// Data types/Touch Probe/E_SignalSource
TYPE E_SignalSource :
 (
	SignalSource_Default,			(* predefined or externally configured *)
	SignalSource_Input1,			(* not selectable in most cases! - digital drive input 1 - from TC 2.11 NC driver 2014 and not TOUCHPROBEMODE_SINGLE_COMPATIBILITYMODE *)
	SignalSource_Input2,			(* not selectable in most cases! - digital drive input 2 - from TC 2.11 NC driver 2014 and not TOUCHPROBEMODE_SINGLE_COMPATIBILITYMODE *)
	SignalSource_Input3,			(* not selectable in most cases! - digital drive input 3 - from TC 2.11 NC driver 2014 and not TOUCHPROBEMODE_SINGLE_COMPATIBILITYMODE *)
	SignalSource_Input4,			(* not selectable in most cases! - digital drive input 4 - from TC 2.11 NC driver 2014 and not TOUCHPROBEMODE_SINGLE_COMPATIBILITYMODE *)
	SignalSource_ZeroPulse := 128,	(* encoder zero pulse. Availability depending on hardware - from TC 2.11 NC driver 2014 and not TOUCHPROBEMODE_SINGLE_COMPATIBILITYMODE *)
	SignalSource_DriveDefined		(* defined by drive parameters - e. g. CAN object 0x60D0 - from TC 2.11 NC driver 2014 and not TOUCHPROBEMODE_SINGLE_COMPATIBILITYMODE *)
 ) UINT;
END_TYPE

// Data types/Touch Probe/E_TouchProbe
(* MC_TouchProbe probes *)
TYPE E_TouchProbe :
 (
	TouchProbe1 := 1,	(* first hardware probe unit with AX2000, SERCOS, KL5xxx and others *)
	TouchProbe2,		(* 2nd probe unit - available from MC_TouchProbe V2 *)
	TouchProbe3,		(* 3rd probe unit - available from MC_TouchProbe V2 *)
	TouchProbe4,		(* 4th probe unit - available from MC_TouchProbe V2 *)
	PlcEvent := 10		(* simple PLC signal TRUE/FALSE *)
 ) UINT;
END_TYPE

// Data types/Touch Probe/E_TouchProbeMode
TYPE E_TouchProbeMode :
 (
	TOUCHPROBEMODE_SINGLE_COMPATIBILITYMODE, (* for TC 2.10 and 2.11 till NC driver 2013 / legacy interface*)
	TOUCHPROBEMODE_SINGLE,			(* multi probe interface - from 2.11 NC driver 2014 / new interface *)
	TOUCHPROBEMODE_CONTINOUS		(* multi probe interface - from 2.11 NC driver 2014 / new interface *)
 ) UINT;
END_TYPE

// Data types/Touch Probe/MC_TouchProbeRecordedData
TYPE MC_TouchProbeRecordedData :
STRUCT
	Counter : LREAL;
	RecordedPosition : LREAL;
	AbsolutePosition	: LREAL;
	ModuloPosition 	: LREAL;
END_STRUCT
END_TYPE

// Data types/Touch Probe/TRIGGER_REF
TYPE TRIGGER_REF :
STRUCT
	EncoderID  		: UDINT;				(* 1..255 *)
	TouchProbe 		: E_TouchProbe;		(* probe unit definition *)
	SignalSource	: E_SignalSource;		(* optional physical signal source used by the probe unit - from TC 2.11 NC driver 2014 with MC_TouchProbe_V2 / no effect for old implementation or TOUCHPROBEMODE_SINGLE_COMPATIBILITYMODE *)
	Edge 			: E_SignalEdge;		(* rising or falling signal edge *)
	(* Mode=TOUCHPROBEMODE_SINGLE as default - changed from TC3 - 2013-04-09 KSt *)
	Mode			: E_TouchProbeMode := TOUCHPROBEMODE_SINGLE; 	(* single shot or continuous monitoring - available from TwinCAT 2.11 NC driver 2014 with MC_TouchProbe_V2 *)
	PlcEvent 		: BOOL;				(* PLC trigger signal input when TouchProbe (probe unit) is set to 'PlcEvent' *)
	ModuloPositions : BOOL;			(* interpretation of FirstPosition, LastPosition and RecordedPosition as modulo positions when TRUE *)
{attribute 'conditionalshow'}
	ProbeState 		: _E_TouchProbeState;	(* internal state of the touch probe sequence *)
END_STRUCT
END_TYPE

// POUs/[Internal]/Objects/_FBAXIS_REF
{attribute 'conditionalshow'}
TYPE _FBAXIS_REF : AXIS_REF;
END_TYPE

// Global Variables/Global_Variables
VAR_GLOBAL
	TcMcGlobal : _TCMCGLOBAL;
END_VAR
VAR_GLOBAL CONSTANT
	DEFAULT_HOME_POSITION 	:	LREAL 	:= 1.0E307;
	DEFAULT_BACKLASHVALUE 	: 	LREAL 	:= 1.0E307;
END_VAR

// Version/Global_Version
{attribute 'TcGenerated'}
{attribute 'no-analysis'}
{attribute 'linkalways'}
// This function has been automatically generated from the project information.
VAR_GLOBAL CONSTANT
	{attribute 'const_non_replaced'}
	stLibVersion_Tc2_MC2 : ST_LibVersion := (iMajor := 3, iMinor := 3, iBuild := 54, iRevision := 0, nFlags := 1, sVersion := '3.3.54.0');
END_VAR

// Data types/Axis Reference/AXIS_REF
(*
	AXIS_REF data structure

	The FBAXIS_REF is actually not a function block but a data structure
	It includes the axis I/O variables as well as additional information.
	The reason for not using a STRUCT is that structures cannot hold
	located I/O variables.
	The user is supposed to use the AXIS_REF data type which internally
	redirects the type to this function block definition (alias).
*)
{attribute 'conditionalshow_all_locals'}
FUNCTION_BLOCK AXIS_REF
VAR_INPUT
	PlcToNc   AT %Q* : PLCTONC_AXIS_REF;
END_VAR
VAR_OUTPUT
	NcToPlc   AT %I* : NCTOPLC_AXIS_REF;
	ADS              : ST_AdsAddress;
	Status           : ST_AxisStatus;
END_VAR
VAR_INPUT
	DriveAddress		: ST_DriveAddress;
END_VAR
VAR
	_internal : _InternalAxisRefData;
	Storage				:	ARRAY [0..127] OF DWORD;	(* universal storage for internal use *)
END_VAR


ReadStatus();

ACTION ReadStatus:
(* NC cycle counter will be incremented after NC task updated the NcToPlc data structure *)
_internal.NcCycleCounter_AtReadStatusCall := SHR(NcToPlc.OpModeDWord, 24);

(* avoid multiple updates during one cycle which would cause additional CPU load *)
IF _internal.NcCycleCounter_AtReadStatusCall <> Status.NcCycleCounter OR _internal.NcCycleCounter_AtReadStatusCall=0 THEN

	(* new cycle - call status function *)
	_internal.LastTaskIndex_AtReadStatusCall := Status.UpdateTaskIndex;

	(* update the axis status
		ForceTaskIndexUpdate makes sure that the index of the current  task will be updated. 
		ForceTaskIndexUpdate=false saves time because a system call to gettaskindex will be avoided.
	*)
	Status := _F_ReadStatus( ForceTaskIndexUpdate:=_internal.CounterSameTaskIndex_AtReadStatusCall<100, NcToPlc := NcToPlc, PlcToNc := PlcToNc, LastStatus:=Status );

	DriveAddress.TcAxisObjectId := _F_GetTcAxisObjectId(AxisId := NcToPlc.AxisId);
	
	(* count number of cycles with the same task index *)
	IF _internal.LastTaskIndex_AtReadStatusCall=Status.UpdateTaskIndex THEN
		IF _internal.CounterSameTaskIndex_AtReadStatusCall<100 THEN
			(* increment counter as long as the update task index does not change - max value is 100 *)
			_internal.CounterSameTaskIndex_AtReadStatusCall := _internal.CounterSameTaskIndex_AtReadStatusCall + 1;
		END_IF
	ELSE
		(* reset counter since update task index has changed - this is not supposed to happen but a user might call ReadStatus in several tasks *)
		_internal.CounterSameTaskIndex_AtReadStatusCall:= 0;
	END_IF
END_IF
END_ACTION

END_FUNCTION_BLOCK

// POUs/[Internal]/_F_ReadStatus
{attribute 'conditionalshow'}
FUNCTION _F_ReadStatus : ST_AxisStatus
VAR_INPUT
	ForceTaskIndexUpdate : BOOL; (* force update of the taskindex with GETCURTASKINDEX - otherwise update only once - 20100416 KSt *)
END_VAR
VAR_IN_OUT
	NcToPlc : NCTOPLC_AXIS_REF;
	PlcToNc : PLCTONC_AXIS_REF;
	LastStatus : ST_AxisStatus;
END_VAR
VAR
	GetTaskIndex : GETCURTASKINDEX;
END_VAR

 (* MOTION CONTROL STATEMACHINE STATES *)
(* no need to initialize since function result is already intialized - 20100416 KSt *)
(*
_F_ReadStatus.ErrorStop			:= FALSE;
_F_ReadStatus.Disabled 			:= FALSE;
_F_ReadStatus.Stopping			:= FALSE;
_F_ReadStatus.StandStill			:= FALSE;
_F_ReadStatus.DiscreteMotion		:= FALSE;
_F_ReadStatus.ContinuousMotion	:= FALSE;
_F_ReadStatus.SynchronizedMotion	:= FALSE;
_F_ReadStatus.Homing			:= FALSE;
*)

_F_ReadStatus.MotionState := _F_AxisState(NcToPlc, PlcToNc);
CASE _F_ReadStatus.MotionState OF
	MC_AXISSTATE_DISABLED :
		_F_ReadStatus.Disabled := TRUE;
	MC_AXISSTATE_STANDSTILL :
		_F_ReadStatus.StandStill := TRUE;
	MC_AXISSTATE_ERRORSTOP :
		_F_ReadStatus.ErrorStop := TRUE;
	MC_AXISSTATE_STOPPING :
		_F_ReadStatus.Stopping := TRUE;
	MC_AXISSTATE_HOMING :
		_F_ReadStatus.Homing	:= TRUE;
	MC_AXISSTATE_DISCRETEMOTION :
		_F_ReadStatus.DiscreteMotion := TRUE;
	MC_AXISSTATE_CONTINOUSMOTION :
		_F_ReadStatus.ContinuousMotion := TRUE;
	MC_AXISSTATE_SYNCHRONIZEDMOTION :
		_F_ReadStatus.SynchronizedMotion := TRUE;
END_CASE

(* NcToPlc.StateDWord *)
_F_ReadStatus.Operational				:= NcToPlc.StateDWord.0;
_F_ReadStatus.Homed				:= NcToPlc.StateDWord.1;		(* homed *)
_F_ReadStatus.NotMoving				:= NcToPlc.StateDWord.2;
_F_ReadStatus.InPositionArea			:= NcToPlc.StateDWord.3;
_F_ReadStatus.inTargetPosition 		:= NcToPlc.StateDWord.4;
_F_ReadStatus.ProtectedMode				:= NcToPlc.StateDWord.5;
_F_ReadStatus.ErrorPropagationDelayed	:= NcToPlc.StateDWord.6;
_F_ReadStatus.HasBeenStopped		:= NcToPlc.StateDWord.7;
_F_ReadStatus.HasJob				:= NcToPlc.StateDWord.8;
_F_ReadStatus.Moving				:= NcToPlc.StateDWord.9 OR NcToPlc.StateDWord.10;
_F_ReadStatus.PositiveDirection		:= NcToPlc.StateDWord.9;
_F_ReadStatus.NegativeDirection 		:= NcToPlc.StateDWord.10;
_F_ReadStatus.HomingBusy			:= NcToPlc.StateDWord.11; 	(* homing *)
_F_ReadStatus.ConstantVelocity 		:= NcToPlc.StateDWord.12;
_F_ReadStatus.Compensating			:= NcToPlc.StateDWord.13;	(* superposition active *)
_F_ReadStatus.ExtSetPointGenEnabled 	:= NcToPlc.StateDWord.14;
_F_ReadStatus.PhasingActive 	:= NcToPlc.StateDWord.15;
_F_ReadStatus.ExternalLatchValid		:= NcToPlc.StateDWord.16;
_F_ReadStatus.NewTargetPosition		:= NcToPlc.StateDWord.17;
_F_ReadStatus.DriveLimitActive 	:= NcToPlc.StateDWord.18; (* 201801213 Fap *)
(*_F_ReadStatus.MovingEndless 		:= NcToPlc.StateDWord.19;	see continuous motion *)
_F_ReadStatus.ControlLoopClosed 		:= NcToPlc.StateDWord.20;
_F_ReadStatus.CamTableQueued 		:= NcToPlc.StateDWord.21;
_F_ReadStatus.CamDataQueued		:= NcToPlc.StateDWord.22;
_F_ReadStatus.CamScalingPending 		:= NcToPlc.StateDWord.23;
_F_ReadStatus.CmdBuffered	 		:= NcToPlc.StateDWord.24;
_F_ReadStatus.PTPmode	 			:= NcToPlc.StateDWord.25;
_F_ReadStatus.SoftLimitMinExceeded	:= NcToPlc.StateDWord.26;
_F_ReadStatus.SoftLimitMaxExceeded	:= NcToPlc.StateDWord.27;
_F_ReadStatus.DriveDeviceError	 	:= NcToPlc.StateDWord.28;
_F_ReadStatus.MotionCommandsLocked	:= NcToPlc.StateDWord.29;
_F_ReadStatus.IoDataInvalid			:= NcToPlc.StateDWord.30;
_F_ReadStatus.Error 					:= NcToPlc.StateDWord.31;

(* NcToPlc.nCoupleState *)
_F_ReadStatus.Coupled		:= NcToPlc.CoupleState > 1;

(* additional status data structue *)
_F_ReadStatus.ErrorID			:= NcToPlc.ErrorCode;
_F_ReadStatus.Accelerating 	:= NcToPlc.AxisState = INT_TO_DWORD(TCNC_PHASE_ACCPOS);
_F_ReadStatus.Decelerating 	:= NcToPlc.AxisState = INT_TO_DWORD(TCNC_PHASE_ACCNEG);

(* axis operation modes *)
_F_ReadStatus.OpMode.PositionAreaMonitoring	:= NcToPlc.OpModeDWord.0;
_F_ReadStatus.OpMode.TargetPositionMonitoring	:= NcToPlc.OpModeDWord.1;
_F_ReadStatus.OpMode.LoopMode				:= NcToPlc.OpModeDWord.2;
_F_ReadStatus.OpMode.MotionMonitoring		:= NcToPlc.OpModeDWord.3;
_F_ReadStatus.OpMode.PEHTimeMonitoring		:= NcToPlc.OpModeDWord.4;
_F_ReadStatus.OpMode.BacklashCompensation	:= NcToPlc.OpModeDWord.5;
_F_ReadStatus.OpMode.DelayedErrorReaction	:= NcToPlc.OpModeDWord.6;	(* 2008-02-20 KSt *)
_F_ReadStatus.OpMode.Modulo				:= NcToPlc.OpModeDWord.7;
_F_ReadStatus.OpMode.SimulationAxis			:= NcToPlc.OpModeDWord.8;	(* 2011-05-31 KSt *)
_F_ReadStatus.OpMode.StopMonitoring			:= NcToPlc.OpModeDWord.12;	(* 2011-12-09 KSt *)
_F_ReadStatus.OpMode.PositionLagMonitoring	:= NcToPlc.OpModeDWord.16;
_F_ReadStatus.OpMode.VelocityLagMonitoring	:= NcToPlc.OpModeDWord.17;
_F_ReadStatus.OpMode.SoftLimitMinMonitoring	:= NcToPlc.OpModeDWord.18;
_F_ReadStatus.OpMode.SoftLimitMaxMonitoring	:= NcToPlc.OpModeDWord.19;
_F_ReadStatus.OpMode.PositionCorrection		:= NcToPlc.OpModeDWord.20;
_F_ReadStatus.OpMode.AllowSlaveCommands	:= NcToPlc.OpModeDWord.21;	(* 2009-02-20 KSt *)
_F_ReadStatus.OpMode.AllowExtSetAxisCommands := NcToPlc.OpModeDWord.22;(* 2011-10-13 KSt *)
(* additional status bits in operation mode dword *)
_F_ReadStatus.NcApplicationRequest			:= NcToPlc.OpModeDWord.23;	(* 2010-04-06 KSt *)

(* NC cycle counter will be incremented after NC task updated the NcToPlc data structure *)
_F_ReadStatus.NcCycleCounter := SHR(NcToPlc.OpModeDWord, 24);

IF 	LastStatus.UpdateTaskIndex=0 OR ForceTaskIndexUpdate THEN
	GetTaskIndex(); (* function call causes high CPU load - supposed to be avoided - 20100416 KSt *)
	_F_ReadStatus.UpdateTaskIndex := GetTaskIndex.index;
	_F_ReadStatus.CycleCounter := TwinCAT_SystemInfoVarList._TaskInfo[_F_ReadStatus.UpdateTaskIndex].cycleCount;
	(*_F_ReadStatus.UpdateCycleTime := TwinCAT_SystemInfoVarList._TaskInfo[_F_ReadStatus.UpdateTaskIndex].cycleTime / LREAL#1.0E6;*)	(* Correction 2009-11-26 KSt *)
	_F_ReadStatus.UpdateCycleTime := TwinCAT_SystemInfoVarList._TaskInfo[_F_ReadStatus.UpdateTaskIndex].cycleTime / LREAL#1.0E7;	(* Correction 2014-05-20 KSt *)
ELSE
	_F_ReadStatus.UpdateTaskIndex := LastStatus.UpdateTaskIndex;
	_F_ReadStatus.CycleCounter := TwinCAT_SystemInfoVarList._TaskInfo[LastStatus.UpdateTaskIndex].cycleCount;
	(*_F_ReadStatus.UpdateCycleTime := TwinCAT_SystemInfoVarList._TaskInfo[LastStatus.UpdateTaskIndex].cycleTime / LREAL#1.0E6;*)	(* Correction 2009-11-26 KSt *)
	_F_ReadStatus.UpdateCycleTime := TwinCAT_SystemInfoVarList._TaskInfo[LastStatus.UpdateTaskIndex].cycleTime / LREAL#1.0E7;	(* Correction 2014-05-20 KSt *)
END_IF

(* 2010-04-26 KSt - Read NC device Info *)
IF TCMCGLOBAL.NcDeviceInfoNcVersion = 0 THEN
	TCMCGLOBAL.ReadDeviceInfo();
END_IF

END_FUNCTION

// POUs/[Internal]/_F_AxisState
{attribute 'conditionalshow'}
(* 	Function returns the current PLCopen axis state *)
(*	see state diagram *)
FUNCTION _F_AxisState : MC_AxisStates

VAR_INPUT
END_VAR
VAR
END_VAR
(*All VAR_IN_OUT variables have been moved to the end of the declaration due to compatibility reasons*)
VAR_IN_OUT
	NcToPlc : NCTOPLC_AXIS_REF;
	PlcToNc : PLCTONC_AXIS_REF;
END_VAR

IF F_AxisInErrorState(NcToPlc.StateDWord) THEN
	IF PlcToNc.ControlDWord.0 THEN
		(* Power.Enable=TRUE but in error state *)
		_F_AxisState := MC_AXISSTATE_ERRORSTOP;
	ELSE
		_F_AxisState := MC_AXISSTATE_DISABLED;
	END_IF
ELSE
(*	IF F_AxisIsReady(NcToPlc.StateDWord) THEN *)			(* 20090205 KSt *)
	IF F_AxisControlLoopClosed(NcToPlc.StateDWord) THEN	(* 20090205 KSt *)
		// IF F_AxisIsCoupled(NcToPlc.CoupleState) THEN (* disabled 20191031 KSt *)
		IF F_AxisIsCoupled(NcToPlc.CoupleState) OR (NOT F_AxisInProtectedMode(NcToPlc.StateDWord) AND NOT F_AxisInPTPmode((NcToPlc.StateDWord))) THEN (* new 20191031 KSt - synchronized motion if axis in other group (NCI, Kinematic etc...) *)
			(* slave or other synchronized group*)
			_F_AxisState := MC_AXISSTATE_SYNCHRONIZEDMOTION;

		ELSIF F_AxisHasJob(NcToPlc.StateDWord) THEN
			(* moving single axis *)
			IF F_AxisHasBeenStopped(NcToPlc.StateDWord) THEN			
				(* axis kept in stop mode by a stop command *)
				_F_AxisState := MC_AXISSTATE_STOPPING;

//				20170206 FAP This will fix the incompatibility to PLCopen state machine using a MC_Halt command 
// 				fix is denied by product management to avoid issues to current users 
//				IF F_AxisMotionCommandsLocked(NcToPlc.StateDWord) THEN
//					(* axis kept in stop mode by a stop command *)
//					_F_AxisState := MC_AXISSTATE_STOPPING;
//				ELSE
//					(* axis kept in discrete motion mode by a halt command *)
//					_F_AxisState := MC_AXISSTATE_DISCRETEMOTION;
//				END_IF
			ELSIF F_AxisIsCalibrating(NcToPlc.StateDWord) THEN
				_F_AxisState := MC_AXISSTATE_HOMING;
			ELSIF F_AxisIsMovingEndless(NcToPlc.StateDWord) THEN
				_F_AxisState := MC_AXISSTATE_CONTINOUSMOTION;
			ELSE
				_F_AxisState := MC_AXISSTATE_DISCRETEMOTION;
			END_IF
		ELSE
			(* ready but no job *)
			IF F_AxisMotionCommandsLocked(NcToPlc.StateDWord) THEN
				(* axis kept in stop mode by a stop command *)
				_F_AxisState := MC_AXISSTATE_STOPPING;
			ELSE
				_F_AxisState := MC_AXISSTATE_STANDSTILL;
			END_IF
		END_IF
	ELSE
		_F_AxisState := MC_AXISSTATE_DISABLED;
	END_IF
END_IF

END_FUNCTION

// POUs/[Internal]/Axis Status Flag Functions/F_AxisInErrorState
{attribute 'conditionalshow'}
FUNCTION F_AxisInErrorState : BOOL
(* 	reference: 	NC -> PLC axis interface (128 bytes)
	check if bit 31 of an axis StateDWord is set:
	Axis is in a fault state
	Achse ist im Fehlerzustand
*)
VAR_INPUT
	StateDWord : DWORD;
END_VAR
VAR
END_VAR

F_AxisInErrorState := (StateDWord AND 2#1000_0000_0000_0000_0000_0000_0000_0000) <> 0;

END_FUNCTION

// POUs/[Internal]/Axis Status Flag Functions/F_AxisIsReady
{attribute 'conditionalshow'}
FUNCTION F_AxisIsReady : BOOL
(* 	reference: 	NC -> PLC axis interface (128 bytes)
	check if bit 0 of an axis StateDWord is set:
	Axis is ready for operation
	Achse ist betriebsbereit
*)
VAR_INPUT
	StateDWord : DWORD;
END_VAR
VAR
END_VAR

F_AxisIsReady := (StateDWord AND 2#0000_0000_0000_0000_0000_0000_0000_0001) <> 0;

END_FUNCTION

// POUs/[Internal]/Axis Status Flag Functions/F_AxisControlLoopClosed
{attribute 'conditionalshow'}
FUNCTION F_AxisControlLoopClosed  : BOOL
(* 	reference: 	NC -> PLC axis interface (128 bytes)
	check if bit 20 of an axis StateDWord is set:
	Axis control loop is closed 
	Achsregelkreis ist geschlossen
*)
VAR_INPUT
	StateDWord : DWORD;
END_VAR
VAR
END_VAR

F_AxisControlLoopClosed := (StateDWord AND 2#0000_0000_0001_0000_0000_0000_0000_0000) <> 0;

END_FUNCTION

// POUs/[Internal]/Axis Status Flag Functions/F_AxisIsCoupled
{attribute 'conditionalshow'}
FUNCTION F_AxisIsCoupled : BOOL
VAR_INPUT
	nCoupleState : DWORD;
END_VAR
VAR
END_VAR

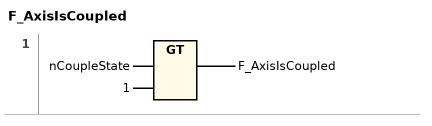
// NETWORK 1
F_AxisIsCoupled := nCoupleState > 1;

END_FUNCTION

// POUs/[Internal]/Axis Status Flag Functions/F_AxisInProtectedMode
{attribute 'conditionalshow'}
FUNCTION F_AxisInProtectedMode  : BOOL
(* 	reference: 	NC -> PLC axis interface (128 bytes)
	check if bit 5 of an axis StateDWord is set:
	Axis is in a protected operating mode (e.g. as a slave axis, or under axis interpolation)
	Achse ist in geschützter Betriebsart (z.B. Slave-Achse oder Achsinterpolation)
*)
VAR_INPUT
	StateDWord : DWORD;
END_VAR
VAR
END_VAR

F_AxisInProtectedMode := (StateDWord AND 2#0000_0000_0000_0000_0000_0000_0010_0000) <> 0;

END_FUNCTION

// POUs/[Internal]/Axis Status Flag Functions/F_AxisInPTPmode
{attribute 'conditionalshow'}
FUNCTION F_AxisInPTPmode : BOOL
(* 	reference: 	NC -> PLC axis interface (128 bytes)
	check if bit 25 of an axis StateDWord is set:
	- The flag signals that the axis accepts PTP motion commands. That requires that the axis is 
	not coupled to other axes and not part of a NC-I or FIFO group.
	- Das Flag zeigt an, dass die Achse PTP Bewegungskommandos entgegen nimmt. Das setzt 
	voraus, dass die Achse nicht gekoppelt ist oder in eine NC-I oder FIFO-Gruppe integriert ist.
*)
VAR_INPUT
	StateDWord : DWORD;
END_VAR
VAR
END_VAR

F_AxisInPTPmode := (StateDWord AND 2#0000_0010_0000_0000_0000_0000_0000_0000) <> 0;

END_FUNCTION

// POUs/[Internal]/Axis Status Flag Functions/F_AxisHasJob
{attribute 'conditionalshow'}
FUNCTION F_AxisHasJob : BOOL
(* 	reference: 	NC -> PLC axis interface (128 bytes)
	check if bit 8 of an axis StateDWord is set:
	Axis has instructions, is carrying instructions out
	Achse hat Auftrag, führt Auftrag aus
*)
VAR_INPUT
	StateDWord : DWORD;
END_VAR
VAR
END_VAR

F_AxisHasJob := (StateDWord AND 2#0000_0000_0000_0000_0000_0001_0000_0000) <> 0;

END_FUNCTION

// POUs/[Internal]/Axis Status Flag Functions/F_AxisHasBeenStopped
{attribute 'conditionalshow'}
FUNCTION F_AxisHasBeenStopped : BOOL
(* 	reference: 	NC -> PLC axis interface (128 bytes)
	check if bit 7 of an axis StateDWord is set:
	Axis has been stopped or is presently executing a stop
	Achse ist gestoppt worden bzw. führt einen Stopp aus
*)
VAR_INPUT
	StateDWord : DWORD;
END_VAR
VAR
END_VAR

F_AxisHasBeenStopped := (StateDWord AND 2#0000_0000_0000_0000_0000_0000_1000_0000) <> 0;

END_FUNCTION

// POUs/Motion/Point To Point Motion/MC_Halt
FUNCTION_BLOCK MC_Halt
(*	This function block commands a controlled motion stop. The axis is moved to
	the state 'DiscreteMotion', until the velocity is zero. With the Done output set, the 
	state is transferred to StandStill.

	Notes:
	- MC_Halt is used to stop the axis under normal operation conditions. 
	  In non-buffered mode it is possible to set another motion command during 
	  deceleration of the axis, which will abort the MC_Halt and will be executed 
	  immediately.
	- If this command is active the next command can be issued. 
	  E.g. a driverless vehicle detects an obstacle and needs to stop. 
	  MC_Halt is issued. Before the standstill is reached the obstacle is 
	  removed and the motion can be continued by setting another motion 
	  command, so the vehicle does not stop.
*)
VAR_IN_OUT
	Axis				:	AXIS_REF; (*Reference to an axis*)
END_VAR
VAR_INPUT
	Execute			:	BOOL;	
	Deceleration		:	LREAL;	
	Jerk				:	LREAL;	
	BufferMode		:	MC_BufferMode;	
	Options			: 	ST_MoveOptions;	 (* optional parameters *)
END_VAR
VAR_OUTPUT
	Done			:	BOOL;	
	Busy			: 	BOOL;	
	Active			: 	BOOL;	
	CommandAborted	:	BOOL;
	Error			:	BOOL;	
{attribute 'displaymode':='hex'}
	ErrorID			:	UDINT;	
END_VAR
VAR
	LastExecutionResult: 	_ST_FunctionBlockResults;
	ADSbusy		: 	BOOL;
	MoveGeneric		: 	_FB_MoveUniversalGeneric;
	CmdNo: UINT;
END_VAR

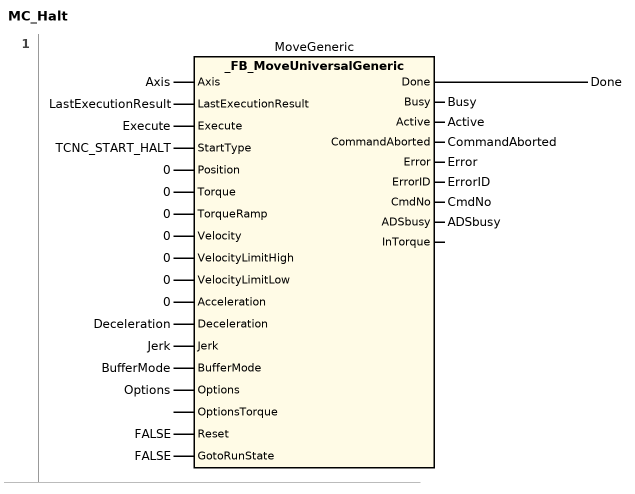
// NETWORK 1
MoveGeneric(
    Axis := Axis,
    LastExecutionResult := LastExecutionResult,
    Execute := Execute,
    StartType := TCNC_START_HALT,
    Position := 0,
    Torque := 0,
    TorqueRamp := 0,
    Velocity := 0,
    VelocityLimitHigh := 0,
    VelocityLimitLow := 0,
    Acceleration := 0,
    Deceleration := Deceleration,
    Jerk := Jerk,
    BufferMode := BufferMode,
    Options := Options,
    Reset := FALSE,
    GotoRunState := FALSE,
    Busy => Busy,
    Active => Active,
    CommandAborted => CommandAborted,
    Error => Error,
    ErrorID => ErrorID,
    CmdNo => CmdNo,
    ADSbusy => ADSbusy); // _FB_MoveUniversalGeneric
Done := MoveGeneric.Done;

END_FUNCTION_BLOCK

// POUs/[Internal]/_FB_MoveUniversalGeneric
{attribute 'conditionalshow'}
FUNCTION_BLOCK _FB_MoveUniversalGeneric
VAR_IN_OUT
	Axis				:	AXIS_REF; (*Reference to an axis*)
	LastExecutionResult: _ST_FunctionBlockResults;
END_VAR
VAR_INPUT
	Execute			:	BOOL;
(*	StartType		: 	UDINT; *)
	StartType		: 	_E_TCNC_StartPosType;	(* 20110511 KSt type changed for Tc3 *)
	Position			:	LREAL;
	Torque				:	LREAL;
	TorqueRamp			:	LREAL;
	Velocity			:	LREAL;
	VelocityLimitHigh	:	LREAL;
	VelocityLimitLow	:	LREAL;
	Acceleration		:	LREAL;
	Deceleration		:	LREAL;
	Jerk				:	LREAL;
(*	Direction			:	MC_Direction := MC_Positive_Direction;	*)(* E *)
	BufferMode		:	MC_BufferMode;
	Options			: 	ST_MoveOptions;
	OptionsTorque	: 	ST_TorqueControlOptions;
	Reset			: 	BOOL;	(* for internal use only *)
	GotoRunState	: 	BOOL;	(* for internal use only *)
	(* FAP 21-02-23 new continuousupdate for torque control *)
	ContinuousUpdate:	BOOL;	(* for internal use only (TorqueControl) *)
END_VAR
VAR_OUTPUT
	Done				:	BOOL;	(* Same meaning as InVelocity for continous motion commands *)
	Busy 				: 	BOOL;
	Active	 			: 	BOOL;
	CommandAborted		:	BOOL;
	Error				:	BOOL;
{attribute 'displaymode':='hex'}
	ErrorID				:	UDINT;
	CmdNo				: 	UINT;
	ADSbusy: BOOL;
	InTorque			: 	BOOL;
END_VAR
VAR
	iState			: 	_E_TcMC_STATES := STATE_INITIALIZATION;
	sStartRequest	:	_ST_TcNC_UnversalAxisStartRequest;
	sTorqueStartRequest	:	_ST_TcNC_UniversalAxisTorqueStartRequest;
	sStartResponse	:	_ST_TcNC_UnversalAxisStartResponse;
	fbAdsReadWrite	: 	ADSRDWRTEX;
	ContinousMode	: 	BOOL;
	InVelocity		: 	BOOL;
	DiffCycleCounter	: 	UDINT;	(* last recent PLC cycle counter difference while Busy *)
END_VAR
VAR
	EmptyStartResponse	: 	_ST_TcNC_UnversalAxisStartResponse;
	COUNT_R			: 	UDINT;
	CounterCmdNoZero	: 	BYTE;
	CounterCmdNotStarted	: 	BYTE;
	DiffCmdNo			: 	INT;
	InitialNcToPlcCmdNo	: 	UINT;
	NcCycleCounter		:	BYTE;
	LastNcCycleCounter	:	BYTE;
	NcMappingCounter 	: 	BYTE;
	NcCycleCounterAvailable: 	BOOL;
	NcCycleCounterNotAvailable: 	BOOL;
	NcCyclicFeedbackExpected: BOOL;
	PlcDebugCode 		: 	DWORD;	(* additional information for debugging purposes will be added to debug messages (ActErrorMessage) *)
	AxisIsSlave			: 	BOOL;
	GetTaskIndex		: 	GETCURTASKINDEX;
	CycleCounter			: 	UDINT;		(* last recent PLC cycle counter while Busy *)
	BusyCounter			: 	UDINT; (* busy cycles since triggering the block - 2018-01-24 KSt *) 
	fbTimeOut			:	TON;
	fbStopMonitoringTimeOut:	TON;
	fbTimeOutMappingCounter :	TON;
	fbOnTrigger			:	R_TRIG;
	sTempMsg			: 	STRING(255);
	AccDecreasing		: BOOL;
	AccOld				: LREAL;

	(* FAP 21-02-23 new continuousupdate for torque control *)
	iContinuousUpdate: BOOL;
END_VAR
VAR CONSTANT
{warning disable C0228}
	OpMode : _ST_TcNc_OperationModes;
{warning restore C0228}
END_VAR

IF NOT _F_TcMC_IsValidAxisRef(Axis) THEN // AXIS REFERENCE CHECK - 2020-09-17 KSt
	Error := TRUE;
	ErrorID := MC_ERROR_INVALIDREFERENCE;
	RETURN;
END_IF

(* ====================================================================== *)
(* *)
(* ====================================================================== *)
IF Reset THEN
	(* Reset FB for internal use only *)
	InTorque := FALSE;
	InVelocity := FALSE;
	Done := FALSE;
	Busy := FALSE;
	Active := FALSE;
	CommandAborted := FALSE;
	Error := FALSE;
	ErrorID := 0;
	fbAdsReadWrite( WRTRD := FALSE );
	iState := STATE_INITIALIZATION;
END_IF

IF Busy THEN
	(* calculate the difference of the PLC cycle counter to check if the function block has been called cyclically while busy *)
	DiffCycleCounter := TwinCAT_SystemInfoVarList._TaskInfo[GetTaskIndex.index].cycleCount - CycleCounter;
	CycleCounter := TwinCAT_SystemInfoVarList._TaskInfo[GetTaskIndex.index].cycleCount;
	BusyCounter := BusyCounter + 1; (* busy cycles since triggering the block - 2018-01-24 KSt *) 
END_IF

fbOnTrigger(CLK:= Execute);

CASE iState OF
STATE_INITIALIZATION:	(* *)
	Busy := FALSE;
	Active := FALSE;
	IF NOT Execute THEN
		Done := FALSE;
		InVelocity := FALSE;	(* KST 2012-05-16 *)
		InTorque := FALSE;
		CommandAborted := FALSE;
		Error := FALSE;			(* reset at falling edge of Execute *)
		ErrorID := 0;
	END_IF
   	IF fbOnTrigger.Q THEN
		(* initialize output values *)
		Done := FALSE;
		InVelocity := FALSE;
		InTorque := FALSE;
		Busy := TRUE;
		BusyCounter := 0; (* busy cycles since triggering the block - 2018-01-24 KSt *) 
		Active := FALSE;
		CommandAborted := FALSE;
		Error := FALSE;
		ErrorID := 0;
		NcCyclicFeedbackExpected := FALSE;
		LastExecutionResult.Done := FALSE;
		LastExecutionResult.CommandAborted := FALSE;
		LastExecutionResult.Error := FALSE;
		LastExecutionResult.ErrorID := 0;
		CounterCmdNoZero := 0;
		CounterCmdNotStarted := 0;
		(*PlcDebugCode := Axis.PlcToNc.Reserved1;*)	(* additional information for debugging purposes will be added to debug messages (ActErrorMessage) *)
		(* nCmdNo := 0; *)
		fbTimeOut(IN:= FALSE);
		fbStopMonitoringTimeOut(IN:= FALSE);
		fbTimeOutMappingCounter(IN:= FALSE);
		fbAdsReadWrite(WRTRD:=FALSE);
		GetTaskIndex();
		CycleCounter := TwinCAT_SystemInfoVarList._TaskInfo[GetTaskIndex.index].cycleCount;
		DiffCycleCounter := 0;
		ActNcCycleCounter(); (* 2014-10-22 KSt *)
		InitialNcToPlcCmdNo := Axis.NcToPlc.CmdNo;

		(* FAP 21-02-23 new continuousupdate for torque control *)
		iContinuousUpdate := ContinuousUpdate;
		
		IF GotoRunState THEN
			(* reset mapping counter *)
			NcMappingCounter := 0;
			LastNcCycleCounter:=DWORD_TO_BYTE(SHR(Axis.NcToPlc.OpModeDWord, 24));
			NcCyclicFeedbackExpected := FALSE;
(*			ActNcCycleCounter();*) (* 2014-10-22 KSt - moved to line above *)
			iState := STATE_RUNNING;
		ELSE
			IF	NOT Axis.NcToPlc.StateDWord.6 (* error delay mode - pass any command during error delay - 2008-11-26 KSt *)
				AND StartType <> TCNC_START_STOPANDLOCK (* no pre-checks for stop and halt - 2008-11-26 KSt *)
				AND StartType<> TCNC_START_HALT (* no pre-checks for stop and halt - 2008-11-26 KSt *)
				THEN
				(* check for error conditions that don't allow to pass a command *)
				IF F_AxisInErrorState(Axis.NcToPlc.StateDWord) THEN
					Error := TRUE;
					ErrorID := Axis.NcToPlc.ErrorCode;
				ELSIF F_AxisInProtectedMode(Axis.NcToPlc.StateDWord) AND ((Axis.NcToPlc.OpModeDWord AND OpMode.AllowSlaveCommands) = 0) THEN (* 2009-02-20 KSt *)
(*				ELSIF F_AxisInProtectedMode(Axis.NcToPlc.StateDWord) THEN *)	 (* 2008-02-20 KSt *)
					(* motion commands on slaves not allowed *)
					Error := TRUE;
					ErrorID := MC_ERROR_AXIS_IN_PROTECTED_MODE;
				(* axisisready is no longer checked by the PLC - 2011-05-31 HKP
				ELSIF NOT F_AxisIsReady(Axis.NcToPlc.StateDWord) THEN
					Error := TRUE;
					ErrorID := MC_ERROR_AXIS_IS_NOT_READY;
				*)
				ELSIF StartType = 0 THEN
					Error := TRUE;
					ErrorID := MC_ERROR_COMMAND_NOT_ALLOWED;
				END_IF
			END_IF
			IF NOT Error THEN (* pass the command to the NC *)
				(* universal axis start *)
				(* fill struct *)
				CASE StartType OF
					TCNC_START_ENDLESS_PLUS,
					TCNC_START_ENDLESS_MINUS,
					TCNC_START_ENDLESSPLUS_SLOWMANUAL,
					TCNC_START_ENDLESSMINUS_SLOWMANUAL,
					TCNC_START_ENDLESSPLUS_FASTMANUAL,
					TCNC_START_ENDLESSMINUS_FASTMANUAL,
					TCNC_START_TORQUE_ABORT,
					TCNC_START_TORQUE_ABSOLUTE,
					TCNC_START_TORQUE_RELATIVE:
						ContinousMode := TRUE;
					ELSE
						(* ContinousMode := FALSE; *)				(* 20100506 KST - changed for MoveContinous Absolute and MoveContinousRelative *)
						ContinousMode := Options.EndVelocity<>0;	(* 20100506 KST - changed for MoveContinous Absolute and MoveContinousRelative *)
				END_CASE
				IF StartType <> TCNC_START_TORQUE_ABORT
				  AND StartType <> TCNC_START_TORQUE_ABSOLUTE 
				  AND StartType <> TCNC_START_TORQUE_RELATIVE THEN
					AxisIsSlave := F_AxisIsCoupled(Axis.NcToPlc.CoupleState);
					sStartRequest.nStartType := StartType;
					sStartRequest.nControlMask := SEL(Options.EnableBlendingPosition, 0, 1);
					sStartRequest.fPosTarget := Position;
					sStartRequest.fVeloRequ := Velocity;
					sStartRequest.fAcc := Acceleration;
					sStartRequest.fDec := Deceleration;
					sStartRequest.fJerk := Jerk;
					sStartRequest.nBufferMode := BufferMode;
					sStartRequest.fBlendingPosition := Options.BlendingPosition;
					sStartRequest.fVeloStart := Options.StartVelocity;
					sStartRequest.fVeloEnd := Options.EndVelocity;
					sStartResponse := EmptyStartResponse;
	
					fbAdsReadWrite.PORT := SEL(AxisIsSlave, AMSPORT_R0_NCSAF, TcMcGlobal.NCPORT_TCMC_COUPLING); (* select SAF port or standard port when coupled *)
					fbAdsReadWrite.PORT := SEL(Axis.ADS.Port = 0, Axis.ADS.port, fbAdsReadWrite.PORT); (* override with user defined port *)
					fbAdsReadWrite.IDXOFFS := SEL(AxisIsSlave,
									TcMcGlobal.Axis.Functions.IDXOFFS.UNIVERSALSTART,			(* standalone axes *)
									TcMcGlobal.Axis.Functions.IDXOFFS.SLAVEUNIVERSALSTART);	(* slave axes with automatic decoupling and succeding universal axis start command *)
					fbAdsReadWrite.IDXOFFS := SEL(F_AxisHasExtSetPointGen(Axis.NcToPlc.StateDWord),
									fbAdsReadWrite.IDXOFFS,
									TcMcGlobal.Axis.Functions.IDXOFFS.EXTSETGENUNIVERSALSTART );	(* 23.11.10: deactivation of external setpoint generator with succeding universal axis start command *)
	
					fbAdsReadWrite(
						NETID:= Axis.ADS.netId,
						IDXGRP:= TcMcGlobal.Axis.Functions.IDXGRP + Axis.NcToPlc.AxisId,
						(* IDXOFFS:= TcMcGlobal.Axis.Functions.IDXOFFS.UNIVERSALSTART, *) (* 24.2.09 KSt - see offset selection above *)
						WRITELEN:= SIZEOF(sStartRequest),
						READLEN:= SIZEOF(sStartResponse),
						SRCADDR:= ADR(sStartRequest),
						DESTADDR:= ADR(sStartResponse),
						WRTRD:= TRUE,
						TMOUT:= TcMcGlobal.tADSTimeOut,
						COUNT_R=> COUNT_R );
	
					iState := STATE_ORDER;
				ELSE
					AxisIsSlave := F_AxisIsCoupled(Axis.NcToPlc.CoupleState);					
					sTorqueStartRequest.nStartType := StartType;
					// 2021-01-19 FAP added additional flag to enable ManualTorqueStartValue
					//sTorqueStartRequest.nControlMask := OptionsTorque.ControlMask;
					sTorqueStartRequest.nControlMask.0 := OptionsTorque.EnableManualTorqueStartValue;
					sTorqueStartRequest.nControlMask.31 := FALSE;
					sTorqueStartRequest.nMode.0 := ContinuousUpdate;
					sTorqueStartRequest.nBufferMode := BufferMode;
					sTorqueStartRequest.fTorque := Torque;
					sTorqueStartRequest.fTorqueRamp := TorqueRamp;				
					sTorqueStartRequest.fVelocityLimitHigh := VelocityLimitHigh;
					sTorqueStartRequest.fVelocityLimitLow := VelocityLimitLow;
					sTorqueStartRequest.fAcceleration := 0; // not implemented
					sTorqueStartRequest.fDeceleration := 0; // not implemented
					sTorqueStartRequest.fManualTorque := OptionsTorque.ManualTorqueStartValue;

					(* FAP 21-02-23 new continuousupdate for torque control *)
					IF iContinuousUpdate THEN
						MEMCPY(destAddr := ADR(Axis.PlcToNc) + 112, srcAddr := ADR(Torque), n:= 8);
					END_IF
					
					sStartResponse := EmptyStartResponse;
	
					fbAdsReadWrite.PORT := SEL(AxisIsSlave, AMSPORT_R0_NCSAF, TcMcGlobal.NCPORT_TCMC_COUPLING); (* select SAF port or standard port when coupled *)
					fbAdsReadWrite.PORT := SEL(Axis.ADS.Port = 0, Axis.ADS.port, fbAdsReadWrite.PORT); (* override with user defined port *)
	
					fbAdsReadWrite(
						NETID:= Axis.ADS.netId,
						IDXGRP:= TcMcGlobal.Axis.Functions.IDXGRP + Axis.NcToPlc.AxisId,
						IDXOFFS := TcMcGlobal.Axis.Functions.IDXOFFS.UNIVERSALTORQUESTART,
						WRITELEN:= SIZEOF(sTorqueStartRequest),
						READLEN:= SIZEOF(sStartResponse),
						SRCADDR:= ADR(sTorqueStartRequest),
						DESTADDR:= ADR(sStartResponse),
						WRTRD:= TRUE,
						TMOUT:= TcMcGlobal.tADSTimeOut,
						COUNT_R=> COUNT_R );
	
					iState := STATE_ORDER;
				END_IF
			END_IF;
		END_IF;
	END_IF;

STATE_ORDER:  (* wait until command is accepted *)
	fbAdsReadWrite(COUNT_R=> COUNT_R );

	(* FAP 21-02-23 new continuousupdate for torque control *)
	IF iContinuousUpdate THEN
		MEMCPY(destAddr := ADR(Axis.PlcToNc) + 112, srcAddr := ADR(Torque), n:= 8);
	END_IF

	IF NOT fbAdsReadWrite.Busy THEN
		IF fbAdsReadWrite.Err OR COUNT_R <> SIZEOF(sStartResponse) THEN
			Error := TRUE;
			ErrorID := fbAdsReadWrite.ErrId;
			ActErrorMessage();
			iState := STATE_INITIALIZATION;
		ELSE
			CmdNo := sStartResponse.nCmdNo;
(*			Active := CmdNo = Axis.NcToPlc.CmdNo;*)	(* 2013-11-22 KSt - removed to avoid Active before next NC mapping has been done after ADS *)
			IF CmdNo <> InitialNcToPlcCmdNo THEN	(* 2014-10-22 KSt *)
				Active := F_AxisHasJob(Axis.NcToPlc.StateDWord) AND (CmdNo = Axis.NcToPlc.CmdNo);	(* 2014-10-22 KSt *)
			END_IF									(* 2014-10-22 KSt *)
			IF Axis.PlcToNc.ControlDWord.29 THEN	(* 2013-10-01 KSt - enabled message with bit 29 (bit 30 still required) *)
				ActErrorMessage();
			END_IF
			(* reset mapping counter *)
			NcMappingCounter := 0;
			LastNcCycleCounter:=DWORD_TO_BYTE(SHR(Axis.NcToPlc.OpModeDWord, 24));
			NcCyclicFeedbackExpected := FALSE;
			ActNcCycleCounter();

			iState := STATE_RUNNING;
		END_IF
	END_IF

STATE_RUNNING:  (* wait until axis stands still *)
	ActNcCycleCounter();
	ActCalcDiffCmdNo();	(* calculate difference between responsed CmdNo and actually running CmdNo *)

	(* FAP 21-02-23 new continuousupdate for torque control *)
	IF iContinuousUpdate THEN
		MEMCPY(destAddr := ADR(Axis.PlcToNc) + 112, srcAddr := ADR(Torque), n:= 8);
		sTorqueStartRequest.fTorque				:= Torque; // FAP 23-02-06 copy new torque input to internal structure for correct value of "InTorque" flag for continuous update mode
	END_IF

	IF CmdNo <> InitialNcToPlcCmdNo THEN		(* 2014-10-22 KSt *)
		Active := sStartResponse.nCmdNo = Axis.NcToPlc.CmdNo;	(* 2014-10-22 KSt *)
	ELSE										(* 2014-10-22 KSt *)
		Active := (sStartResponse.nCmdNo = Axis.NcToPlc.CmdNo) AND NcCyclicFeedbackExpected; (* 2013-07-10 KSt *)
	END_IF										(* 2014-10-22 KSt *)
	
	IF Axis.NcToPlc.AxisState=INT_TO_DWORD(TCNC_PHASE_EXTSETGEN_MODE1) AND NcCyclicFeedbackExpected THEN	(* 20140801 KSt check for external set point generator added *)
		(* if the external set point generator has been enabled *)
		CommandAborted := TRUE;
		iState := STATE_INITIALIZATION;

	ELSIF Active THEN
		(* command is active and the axis motion status must be monitored *)
		IF (StartType=TCNC_START_STOPANDLOCK) OR (StartType=TCNC_START_HALT) THEN
			ActMonitorStop(); 			(* used with MC_Halt and MC_Stop *)
		ELSIF ContinousMode THEN
			IF StartType <> TCNC_START_TORQUE_ABORT
			  AND StartType <> TCNC_START_TORQUE_ABSOLUTE 
			  AND StartType <> TCNC_START_TORQUE_RELATIVE THEN
				ActMonitorContinousMotion(); (* used with e. g. MoveVelocity *)
			ELSIF StartType = TCNC_START_TORQUE_ABORT THEN
				ActMonitorAbortTorque(); (* used with AbortTorqueControl *)
			ELSE
				ActMonitorContinuousTorque(); (* used with TorqueControl *)
			END_IF
		ELSE
			ActMonitorDiscreteMotion();	(* used with e. g. MoveAbsolute *)
		END_IF

		(* FAP 21-02-23 new continuousupdate for torque control *)
		IF iContinuousUpdate THEN
			IF TorqueRamp <> sTorqueStartRequest.fTorqueRamp
			  OR VelocityLimitHigh <> sTorqueStartRequest.fVelocityLimitHigh
			  OR VelocityLimitLow <> sTorqueStartRequest.fVelocityLimitLow THEN
			  	sTorqueStartRequest.fTorqueRamp			:= TorqueRamp;
				sTorqueStartRequest.fVelocityLimitHigh	:= VelocityLimitHigh;
				sTorqueStartRequest.fVelocityLimitLow	:= VelocityLimitLow;
				sTorqueStartRequest.nControlMask.31		:= TRUE;
				fbAdsReadWrite(WRTRD:= FALSE);
				fbAdsReadWrite(WRTRD:= TRUE);
				
				iState := STATE_ORDER;		  
			END_IF
		END_IF
		
	// ELSIF (* command not yet active *)
	ELSIF NcCyclicFeedbackExpected THEN (* command not yet active - 20171218 KSt NcCyclicFeedbackExpected added *)
		IF F_AxisIsCoupled(Axis.NcToPlc.CoupleState) THEN	(* 20090205 KSt *)
			(* if axis is coupled during motion (FlyingSaw) all commands are aborted - 20090205 KSt*)
			CommandAborted := TRUE;
			iState := STATE_INITIALIZATION;
		// ELSIF Axis.NcToPlc.CmdNo = 0 AND NcCyclicFeedbackExpected THEN  				(* 20090206 KSt *)
		ELSIF Axis.NcToPlc.CmdNo = 0 THEN  												(* 2017-12-18 KSt *)
			CounterCmdNoZero := CounterCmdNoZero + 1;
			IF CounterCmdNoZero > TcMcGlobal.NCTOPLC_FEEDBACK_MAXWAITCYCLES THEN (* wait for a certain number of cycles before error *)
				(* CmdNo zero is not supposed to happen - it may come up after a coupling situation for a few cycles *)
				Error := TRUE;
				ErrorID := MC_ERROR_BUFFERED_COMMAND_CMDNOZERO; (* no command state feedback from NC *)
				iState := STATE_INITIALIZATION;
			END_IF
		ELSIF DiffCmdNo=1 THEN (* running command number is 1 higher than expected *) (* 20110421 KSt *)
			(* feedback CmdNo is exactly ONE increment higher than my command *)
			(* command was aborted or successfully finished *)
			Error := GETBIT32(Axis.NcToPlc.CmdState, INT_TO_SINT(CMDSTATE_LASTCMD_ENDED_WITH_ERROR));
			CommandAborted := NOT Error AND GETBIT32(Axis.NcToPlc.CmdState, INT_TO_SINT(CMDSTATE_LASTCMD_ABORTED_WITHOUT_ERROR));
			Done := NOT Error AND NOT CommandAborted AND GETBIT32(Axis.NcToPlc.CmdState, INT_TO_SINT(CMDSTATE_LASTCMD_SUCCESSFULLY_EXECUTED));	(* 20100514 KSt *)
			IF Error THEN
				(* if axis error-Id is valid then feed it back - otherwhise errror-Id is unknown. *)
				ErrorID := SEL(Axis.NcToPlc.ErrorCode=0, Axis.NcToPlc.ErrorCode, MC_ERROR_BUFFERED_COMMAND_ERRORID_NOT_AVAILABLE );
			END_IF
			IF NOT Done AND NOT CommandAborted AND NOT Error THEN
				Error := TRUE;
				ErrorID := MC_ERROR_BUFFERED_COMMAND_NO_STATE_FEEDBACK; (* no command state feedback from NC *)
			END_IF
			iState := STATE_INITIALIZATION;
		ELSIF DiffCmdNo=2 THEN (* running command number is 2 higher than expected *) (* 20110421 KSt *)
			(* feedback CmdNo is exactly TWO increments higher than my command  - 20090116 KSt *)
			Error := GETBIT32(Axis.NcToPlc.CmdState, INT_TO_SINT(CMDSTATE_LASTCMD_ENDED_WITH_ERROR)); (* error of command+1 *)
			(* if command+1 was aborted then this command has been aborted as well *)
			CommandAborted := NOT Error AND GETBIT32(Axis.NcToPlc.CmdState, INT_TO_SINT(CMDSTATE_LASTCMD_ABORTED_WITHOUT_ERROR));
			IF NOT CommandAborted THEN
				(* if previous command has not been aborted - the status of this command is unknown *)
				Error := TRUE;	(* command monitoring not possible; probably because function block was not called cyclically *)
				ErrorID := SEL( DiffCycleCounter > 1, MC_ERROR_BUFFERED_COMMAND_MONITORING_IMPOSSIBLE, MC_ERROR_BUFFCMD_MONITRNGIMPOSS_FBNOTCALLEDCYC);	(* additional error code with command aborted - command monitoring impossible because the block is not called cyclically - 2011-08-01 KSt *)
			END_IF
			iState := STATE_INITIALIZATION;
		ELSIF DiffCmdNo > 0 THEN (* running command number is 3 or more higher than expected *) (* 20110421 KSt *)
			(* feedback CmdNo is THREE or more increments higher than my command *)
			(* command was aborted - command monitoring impossible *)
			Error := TRUE; 	(* command monitoring not possible; probably because function block was not called cyclically *)
			ErrorID := SEL( DiffCycleCounter > 1, MC_ERROR_BUFFERED_COMMAND_MONITORING_IMPOSSIBLE, MC_ERROR_BUFFCMD_MONITRNGIMPOSS_FBNOTCALLEDCYC); (* additional error code with command aborted - command monitoring impossible because the block is not called cyclically - 2011-08-01 KSt *)
			(*CommandAborted := TRUE;*)	(*  20090116 KSt *)
			iState := STATE_INITIALIZATION;
		ELSIF F_AxisInErrorState(Axis.NcToPlc.StateDWord) THEN
			(* axis error came up before this command has been started *)
			Error := TRUE;
			ErrorID := AXIS.NcToPlc.ErrorCode;
			iState := STATE_INITIALIZATION;
		// ELSIF NOT F_AxisHasJob(Axis.NcToPlc.StateDWord) AND NcCyclicFeedbackExpected THEN (* 2017-12-18 KSt NcCyclicFeedbackExpected removed *)
		ELSIF NOT F_AxisHasJob(Axis.NcToPlc.StateDWord) THEN
			(* CmdNo is still lower than my command - command has not been initiated *)
			IF F_AxisHasBeenStopped(Axis.NcToPlc.StateDWord) THEN
				CommandAborted := TRUE;		(* stopp command aborts this command *)
				iState := STATE_INITIALIZATION;
			ELSE
				(* other cases are not supposed to happen and are error conditions *)
				CounterCmdNotStarted := CounterCmdNotStarted + 1;
				IF CounterCmdNotStarted > TcMcGlobal.NCTOPLC_FEEDBACK_MAXWAITCYCLES THEN (* wait for a certain number of cycles before error *)
					Error := TRUE;
					ErrorID := MC_ERROR_BUFFERED_COMMAND_NOT_STARTED; (* reason unknown *)
					iState := STATE_INITIALIZATION;
				END_IF
			END_IF
			(* timeout check *);
		END_IF
		IF (Error OR CommandAborted) AND (iState<>STATE_RUNNING) THEN
			ActErrorMessage();
		END_IF
	END_IF

ELSE  (* CASE : Unknown program state *)
	iState:= STATE_INITIALIZATION;
END_CASE

ADSbusy := fbAdsReadWrite.BUSY;
IF iState=STATE_INITIALIZATION THEN
	(* reset Busy immediately  when sequence ends *)
	IF Busy THEN
		LastExecutionResult.Done := Done;
		LastExecutionResult.CommandAborted := CommandAborted;
		LastExecutionResult.Error := Error;
		LastExecutionResult.ErrorID := ErrorID;
		LastExecutionResult.BusyCounter := BusyCounter; (* busy cycles since triggering the block - 2018-01-24 KSt *) 
	END_IF
	Busy := FALSE;
	Active := FALSE;
END_IF

ACTION ActCalcDiffCmdNo:
(* 20110421 KSt *)
(* calculate the difference between the responsed CmdNo and the actually running CmdNo *)
IF sStartResponse.nCmdNo = 0 OR Axis.NcToPlc.CmdNo = 0 THEN
	DiffCmdNo := -16#8000;	(* special invalid case - feedback is maximum negative difference *)
ELSIF sStartResponse.nCmdNo > 16#A000 AND Axis.NcToPlc.CmdNo < 16#4000 THEN
	(* overrun - running CmdNo is higher than the responded number *)
	DiffCmdNo := WORD_TO_INT(Axis.NcToPlc.CmdNo - sStartResponse.nCmdNo - 1);	(* substract -1 because 0 is an invalid command number *)
ELSIF sStartResponse.nCmdNo < 16#4000 AND Axis.NcToPlc.CmdNo > 16#A000 THEN
	(* overrun - running CmdNo is lower than the responded number *)
	DiffCmdNo := WORD_TO_INT(Axis.NcToPlc.CmdNo - sStartResponse.nCmdNo + 1);	(* add 1 because 0 is an invalid command number *)
ELSE
	DiffCmdNo := WORD_TO_INT(Axis.NcToPlc.CmdNo - sStartResponse.nCmdNo);
END_IF
END_ACTION

ACTION ActErrorMessage:
IF Axis.PlcToNc.ControlDWord.30 THEN (* bit 30 - debug mode enabled *)
	(* FEHLERMELDUNG *)
	sTempMsg	:= 'TCMC:UAS Axis '; 	(* UAS = universal axis start *)
	sTempMsg	:= CONCAT( sTempMsg, UDINT_TO_STRING( Axis.NcToPlc.AxisId ) );
	sTempMsg	:= CONCAT( sTempMsg, ', CmdNo: ' );
	sTempMsg	:= CONCAT( sTempMsg, UDINT_TO_STRING( sStartResponse.nCmdNo ) );
	IF Error THEN
		sTempMsg	:= CONCAT( sTempMsg, ', Error: 0x' );
		sTempMsg	:= CONCAT( sTempMsg, _F_TcMC_DWORD_TO_HEXSTR(ErrorID) );
	END_IF
	IF CommandAborted THEN
		sTempMsg	:= CONCAT( sTempMsg, ', ABORTED ' );
	END_IF
	sTempMsg	:= CONCAT( sTempMsg, ', StartType: ' );
	IF StartType <> TCNC_START_TORQUE_ABORT
	  AND StartType <> TCNC_START_TORQUE_ABSOLUTE 
	  AND StartType <> TCNC_START_TORQUE_RELATIVE THEN
		sTempMsg	:= CONCAT( sTempMsg, UDINT_TO_STRING( sStartRequest.nStartType ) );
	ELSE
		sTempMsg	:= CONCAT( sTempMsg, UDINT_TO_STRING( sTorqueStartRequest.nStartType ) );	
	END_IF
	sTempMsg	:= CONCAT( sTempMsg, ', SetPos: ' );
	sTempMsg	:= CONCAT( sTempMsg, LREAL_TO_STRING( _F_TcMC_Round( Axis.NcToPlc.SetPos , 4) ) );
	sTempMsg	:= CONCAT( sTempMsg, ', SetVelo: ' );
	sTempMsg	:= CONCAT( sTempMsg, LREAL_TO_STRING( _F_TcMC_Round( Axis.NcToPlc.SetVelo, 4) ) );
	sTempMsg	:= CONCAT( sTempMsg, ', SetAcc: ' );
	sTempMsg	:= CONCAT( sTempMsg, LREAL_TO_STRING( _F_TcMC_Round( Axis.NcToPlc.SetAcc, 4) ) );
	IF StartType <> TCNC_START_TORQUE_ABORT
	  AND StartType <> TCNC_START_TORQUE_ABSOLUTE 
	  AND StartType <> TCNC_START_TORQUE_RELATIVE THEN
		sTempMsg	:= CONCAT( sTempMsg, ', PosTarget: ' );
		sTempMsg	:= CONCAT( sTempMsg, LREAL_TO_STRING( _F_TcMC_Round( sStartRequest.fPosTarget, 4) ) );
		sTempMsg	:= CONCAT( sTempMsg, ',  VeloRequ: ' );
		sTempMsg	:= CONCAT( sTempMsg, LREAL_TO_STRING( _F_TcMC_Round(sStartRequest.fVeloRequ, 4) ) );
		sTempMsg	:= CONCAT( sTempMsg, ',  Acc: ' );
		sTempMsg	:= CONCAT( sTempMsg, LREAL_TO_STRING( _F_TcMC_Round( sStartRequest.fAcc, 4) ) );
		sTempMsg	:= CONCAT( sTempMsg, ',  Dec: ' );
		sTempMsg	:= CONCAT( sTempMsg, LREAL_TO_STRING( _F_TcMC_Round( sStartRequest.fDec, 4) ) );
		sTempMsg	:= CONCAT( sTempMsg, ',  Jerk: ' );
		sTempMsg	:= CONCAT( sTempMsg, LREAL_TO_STRING( _F_TcMC_Round( sStartRequest.fJerk, 4) ) );
		sTempMsg	:= CONCAT( sTempMsg, ', BufMode: ' );
		sTempMsg	:= CONCAT( sTempMsg, UDINT_TO_STRING(sStartRequest.nBufferMode ) );
		sTempMsg	:= CONCAT( sTempMsg, ',  BlendPos: ' );
		sTempMsg	:= CONCAT( sTempMsg, LREAL_TO_STRING( _F_TcMC_Round( sStartRequest.fBlendingPosition, 4) ) );
	ELSE
		sTempMsg	:= CONCAT( sTempMsg, ', Torque: ' );
		sTempMsg	:= CONCAT( sTempMsg, LREAL_TO_STRING( _F_TcMC_Round( sTorqueStartRequest.fTorque, 4) ) );
		sTempMsg	:= CONCAT( sTempMsg, ', TorqueRamp: ' );
		sTempMsg	:= CONCAT( sTempMsg, LREAL_TO_STRING( _F_TcMC_Round( sTorqueStartRequest.fTorqueRamp, 4) ) );
		sTempMsg	:= CONCAT( sTempMsg, ',  VeloHigh: ' );
		sTempMsg	:= CONCAT( sTempMsg, LREAL_TO_STRING( _F_TcMC_Round(sTorqueStartRequest.fVelocityLimitHigh, 4) ) );
		sTempMsg	:= CONCAT( sTempMsg, ',  VeloLow: ' );
		sTempMsg	:= CONCAT( sTempMsg, LREAL_TO_STRING( _F_TcMC_Round(sTorqueStartRequest.fVelocityLimitLow, 4) ) );
		sTempMsg	:= CONCAT( sTempMsg, ',  Acc: ' );
		sTempMsg	:= CONCAT( sTempMsg, LREAL_TO_STRING( _F_TcMC_Round( sTorqueStartRequest.fAcceleration, 4) ) );
		sTempMsg	:= CONCAT( sTempMsg, ',  Dec: ' );
		sTempMsg	:= CONCAT( sTempMsg, LREAL_TO_STRING( _F_TcMC_Round( sTorqueStartRequest.fDeceleration, 4) ) );
		sTempMsg	:= CONCAT( sTempMsg, ', BufMode: ' );
		sTempMsg	:= CONCAT( sTempMsg, UDINT_TO_STRING(sTorqueStartRequest.nBufferMode ) );
	END_IF
	sTempMsg	:= CONCAT( sTempMsg, ',  ADS-Stamp: ' );
	sTempMsg	:= CONCAT( sTempMsg, UDINT_TO_STRING( fbAdsReadWrite.fbAdsRdWrt.STAMP_I) );

	(* additional PLC debug info for Beckhoff debugging programs *)
	(*
	IF Axis.PlcToNc.Reserved1 <> 0 THEN
		sTempMsg 	:= CONCAT( sTempMsg, ', PLC-Code=' );
		sTempMsg 	:= CONCAT( sTempMsg, DWORD_TO_STRING(PlcDebugCode) );
	END_IF
	*)
	IF Error THEN
		ADSLOGSTR( ADSLOG_MSGTYPE_ERROR + ADSLOG_MSGTYPE_LOG, sTempMsg, '' );		(* vom Typ <Fehlermeldung> *)
	ELSIF CommandAborted THEN
		ADSLOGSTR( ADSLOG_MSGTYPE_WARN, sTempMsg, '' ); 		(* vom Typ <Warnungsmeldung> *)
	ELSE
		ADSLOGSTR( ADSLOG_MSGTYPE_HINT, sTempMsg, '' ); 			(* vom Typ <Hinweismeldung> *)
	END_IF
END_IF
END_ACTION

ACTION ActMonitorAbortTorque:
(*
 * 	monitor a abort torque control
 *
 *	monitor until the set torque derivative is zero 
 * 	used with MC_AbortTorqueControl command
*)

(* error while in motion *)
IF	F_AxisInErrorState(Axis.NcToPlc.StateDWord) THEN
	Error := TRUE;
	ErrorID := Axis.NcToPlc.ErrorCode;
	iState := STATE_INITIALIZATION;

(* check for end of torque control  *)
ELSIF Axis.NcToPlc.SetTorqueDerivative = 0 THEN
	(* axis has stopped torque control *)
	Done := TRUE;
	iState := STATE_INITIALIZATION;
END_IF;
END_ACTION

ACTION ActMonitorContinousMotion:
(*
 * 	monitor continous motion
 *
 * 	monitor UNTIL the axis is in velocity AND the Execute-Input is FALSE
 * 	used with MoveVelocity and other continous commands
*)
IF F_AxisInErrorState(StateDWord := Axis.NcToPlc.StateDWord) THEN (* error while positioning *)
	Error := TRUE;
	ErrorID := Axis.NcToPlc.ErrorCode;
	InVelocity := FALSE;	(* reset InVelocity in case of error or abortion - KST 2012-05-16 *)
	iState := STATE_INITIALIZATION;
ELSIF NOT F_AxisHasJob(Axis.NcToPlc.StateDWord) OR F_AxisHasBeenStopped(Axis.NcToPlc.StateDWord) THEN (* KSt 27.5.03 *)
	(* aborted during accelertion *)
	CommandAborted := TRUE;
	InVelocity := FALSE;	(* reset InVelocity in case of error or abortion - KST 2012-05-16 *)
	iState := STATE_INITIALIZATION;
ELSIF InVelocity AND NOT Execute THEN
	(* end of axis control after beeing in velocity for at least one cycle *)
	iState := STATE_INITIALIZATION;
(* ELSIF Axis.NcToPlc.AxisState = TCNC_PHASE_VELOCONST THEN *)	(* 20100506 KST - changed for MoveContinous Absolute and MoveContinousRelative *)
(*ELSIF Axis.NcToPlc.AxisState = INT_TO_DWORD(TCNC_PHASE_VELOCONST) AND F_AxisIsMovingEndless(Axis.NcToPlc.StateDWord) THEN*)	(* 20100506 KST - changed for MoveContinous Absolute and MoveContinousRelative *)
ELSIF F_AxisIsMovingEndless(Axis.NcToPlc.StateDWord)	(* 20100506 KST - changed for MoveContinous Absolute and MoveContinousRelative *)
	AND ((Axis.NcToPlc.AxisState = INT_TO_DWORD(TCNC_PHASE_VELOCONST)) OR	(* continous axes *)
		   (Axis.NcToPlc.AxisState = INT_TO_DWORD(TCNC_PHASE_TWOSPEED_MOVING)) AND F_AxisReachedConstantVelocity(Axis.NcToPlc.StateDWord)) (* 20110719 KST - two speed axes *)
	THEN
	InVelocity := TRUE;
ELSIF InVelocity AND NOT F_AxisIsCompensating(Axis.NcToPlc.StateDWord) THEN
	(* axis was InVelocity but isn't any more, superposition is allowed but *)
	(* any other reason is an abortion *)
	CommandAborted := TRUE;
	InVelocity := FALSE;	(* reset InVelocity in case of error or abortion - KST 2012-05-16 *) 
	iState := STATE_INITIALIZATION;
END_IF
Done := InVelocity;
END_ACTION

ACTION ActMonitorContinuousTorque:
(*
 * 	monitor continuous torque control
 *
 * 	monitor UNTIL the axis is in torque AND the Execute-Input is FALSE
 * 	used with TorqueControl command
*)

(* FAP 2020-12-04 observing flag directly from axis interface and compare difference to 1E-6 instead of direct compare *)
InTorque := NOT F_AxisDriveLimitActive(Axis.NcToPlc.StateDWord)
			AND ABS(Axis.NcToPlc.SetTorqueDerivative) < 1E-6
			AND ABS(Axis.NcToPlc.SetTorque - sTorqueStartRequest.fTorque) < 1E-6;

IF F_AxisInErrorState(StateDWord := Axis.NcToPlc.StateDWord) THEN (* error while positioning *)
	Error := TRUE;
	ErrorID := Axis.NcToPlc.ErrorCode;
	InTorque := FALSE;	(* reset InTorque in case of error or abortion *)
	iState := STATE_INITIALIZATION;
ELSIF NOT F_AxisHasJob(Axis.NcToPlc.StateDWord) OR F_AxisHasBeenStopped(Axis.NcToPlc.StateDWord) THEN
	(* aborted during accelertion *)
	CommandAborted := TRUE;
	InTorque := FALSE;	(* reset InTorque in case of error or abortion*)
	iState := STATE_INITIALIZATION;
ELSIF InTorque AND NOT Execute THEN
	(* end of axis control after beeing in torque for at least one cycle *)
	iState := STATE_INITIALIZATION;
END_IF
END_ACTION

ACTION ActMonitorDiscreteMotion:
(*
 * 	monitor discrete motion 
 *
 *	monitor until the target position is reached 
 * 	used with MC_MoveAbsolute and other discrete commands
*)

(* check for reached target position *)
// IF (Axis.NcToPlc.OpModeDWord AND  OpMode.TargetPosControl) > 0 THEN (* Target position controlling and PEH enabled ? *)
IF NOT Options.IgnorePositionMonitoring AND ((Axis.NcToPlc.OpModeDWord AND OpMode.TargetPosControl) > 0) THEN (* Target position controlling and PEH enabled ? *) // 20190311 Ignore flag added
	IF NOT F_AxisHasJob(Axis.NcToPlc.StateDWord) AND F_AxisIsAtTargetPosition(Axis.NcToPlc.StateDWord) THEN
		Done := TRUE;
		iState := STATE_INITIALIZATION;
	END_IF
ELSE
	// IF (Axis.NcToPlc.OpModeDWord AND OpMode.PosAreaControl) > 0 THEN (* Target position controlling enabled ? *)
	IF NOT Options.IgnorePositionMonitoring AND ((Axis.NcToPlc.OpModeDWord AND OpMode.PosAreaControl) > 0) THEN (* Target position controlling enabled ? *)	// 20190311 Ignore flag added
		IF NOT F_AxisHasJob(Axis.NcToPlc.StateDWord) AND F_AxisInPositionWindow(Axis.NcToPlc.StateDWord) THEN
			Done := TRUE;
			iState := STATE_INITIALIZATION;
		END_IF
	ELSE
		IF NOT F_AxisHasJob(Axis.NcToPlc.StateDWord) THEN
			Done := TRUE;
			iState := STATE_INITIALIZATION;
		END_IF
	END_IF
END_IF;
(* check for timeout *)
IF NOT done AND NOT F_AxisHasJob(Axis.NcToPlc.StateDWord) THEN
	fbTimeOut(IN:= TRUE, PT:= TcMcGlobal.tTargetPosTimeOut);
	IF fbTimeOut.Q THEN
		Error := TRUE;
		ErrorID := MC_ERROR_TARGETPOS_TIMEOUT;
		iState := STATE_INITIALIZATION;
	END_IF;
END_IF;

(* error while positioning *)
IF	F_AxisInErrorState(Axis.NcToPlc.StateDWord) THEN
	Done := FALSE;	(* KSt - 2013-05-23 *)
	Error := TRUE;
	ErrorID := Axis.NcToPlc.ErrorCode;
	iState := STATE_INITIALIZATION;
ELSIF 	F_AxisHasBeenStopped(Axis.NcToPlc.StateDWord)
		AND NOT F_AxisHasJob(Axis.NcToPlc.StateDWord)
		AND NOT (StartType=TCNC_START_HALT)
		AND NOT (StartType=TCNC_START_STOPANDLOCK)
		THEN
		(* manual stop or stop FB ? *)
		Done := FALSE;	(* KSt - 2013-07-02 - reset Done in case of CommandAborted *)
(*		ErrorID := MC_ERROR_AXIS_HAS_BEEN_STOPPED;*)	(* HKP - 2013-07-02 - ErrorID removed because just informational feedback *)
		CommandAborted 	:= TRUE;
		iState := STATE_INITIALIZATION;
(*	bit 18 is not implemented - 20080610 KSt
ELSIF  F_AxisIsNotInTargetPosition(Axis.NcToPlc.StateDWord) THEN
	( target pos can NOT be reached )
		ErrorID := MC_ERROR_TARGETPOS_TIMEOUT;
		Error := TRUE;
		iState := STATE_INITIALIZATION;
*)
END_IF
END_ACTION

ACTION ActMonitorStop:
(*
 * 	monitor a motion stop or halt
 *
 *	monitor until the target position is reached 
 * 	used with MC_Halt and MC_Stop commands
*)
(* FAP 2019-09-13 Check if acc is decreasing for stopping with very low dynamics in accelerating phase *)
AccDecreasing := (AccOld - ABS(Axis.NcToPlc.SetAcc)) > 0.0 AND Axis.NcToPlc.AxisState = INT_TO_DWORD(TCNC_PHASE_ACCPOS);
AccOld := ABS(Axis.NcToPlc.SetAcc);

(* check for deceleration *)
(* fbTimeOut(IN:= Axis.NcToPlc.AxisState <> INT_TO_DWORD(TCNC_PHASE_ACCNEG), PT:= TcMcGlobal.tTargetPosTimeOut);*)

(* check for deceleration or decreasing acceleration (FAP 2019-09-13) *)
fbTimeOut(IN:= Axis.NcToPlc.AxisState <> INT_TO_DWORD(TCNC_PHASE_ACCNEG) AND NOT AccDecreasing, PT:= TcMcGlobal.tTargetPosTimeOut);
fbStopMonitoringTimeOut();

(* error while positioning *)
IF	F_AxisInErrorState(Axis.NcToPlc.StateDWord) THEN
	Error := TRUE;
	ErrorID := Axis.NcToPlc.ErrorCode;
	iState := STATE_INITIALIZATION;

(* check for end of motion  *)
ELSIF NOT F_AxisHasJob(Axis.NcToPlc.StateDWord) THEN
	IF F_AxisIsAtTargetPosition(Axis.NcToPlc.StateDWord) THEN
		(* axis is in standstill and the actual value is inside the monitoring window *)
		Done := TRUE;
		iState := STATE_INITIALIZATION;
	ELSIF Options.IgnorePositionMonitoring OR ((Axis.NcToPlc.OpModeDWord AND OpMode.StopMonitoring) = 0) THEN (* stop monitoring inactiv *)
		(* done after has job false without other monitoring *)
		Done := TRUE;
		iState := STATE_INITIALIZATION;
	ELSIF Options.EnableStopPositionMonitoring AND ((Axis.NcToPlc.OpModeDWord AND OpMode.StopMonitoring) > 0) AND TcMcGlobal.NcDeviceInfoNcVersion >= 16#03011194 (* NC 4500 *) THEN // if StopPositionMonitoring is enabled from TC3.1 4024 - 20191010 KSt
		IF fbTimeOut.Q THEN // if StopPositionMonitoring is enabled, timeout after 6 seconds (from TC3.1 4024) - 20191010 KSt 
			Error := TRUE;
			ErrorID := MC_ERROR_TARGETPOS_TIMEOUT;
			iState := STATE_INITIALIZATION;
		END_IF
	ELSE
		(* 20111208 KSt - if stop monitoring is active, axis waits for actual position beeing in target window *)
		fbStopMonitoringTimeOut(IN:= TRUE, PT:= TcMcGlobal.tStopMonitoringTimeOut);	(* start monitoring timer *)
		IF fbStopMonitoringTimeOut.Q THEN (* not error but end of monitoring *)
			(* axis set position is in standstill but the acutal value did probalby not reach the monitoring window - no error in this case *)
			Done := TRUE;
			iState := STATE_INITIALIZATION;
 		END_IF
	END_IF
	
(* old code before 2019-10 - substitued by code block above
	// IF 	(Axis.NcToPlc.OpModeDWord AND OpMode.StopMonitoring) > 0 THEN	(* stop monitoring active *)
	IF NOT Options.IgnorePositionMonitoring AND ((Axis.NcToPlc.OpModeDWord AND OpMode.StopMonitoring) > 0) THEN	(* stop monitoring active *) // 20190311 Ignore flag added
		(* 20111208 KSt - if stop monitoring is active, axis waits for actual position beeing in target window *)
		fbStopMonitoringTimeOut(IN:= TRUE, PT:= TcMcGlobal.tStopMonitoringTimeOut);	(* start monitoring timer *)
		IF F_AxisIsAtTargetPosition(Axis.NcToPlc.StateDWord) THEN
			(* axis is in standstill and the actual value is inside the monitoring window *)
			Done := TRUE;
			iState := STATE_INITIALIZATION;
		ELSIF  fbStopMonitoringTimeOut.Q THEN (* not error but end of monitoring *)
			IF TcMcGlobal.NcDeviceInfoNcVersion >= 16#03011194  (* NC 4500 *) THEN // Error instead of Done from TC 3.1.4500 - 20190311
				Error := TRUE;
				ErrorID := MC_ERROR_TARGETPOS_TIMEOUT;
				iState := STATE_INITIALIZATION;
			ELSE // no error with previous NC driver versions
				(* axis set position is in standstill but the acutal value did probalby not reach the monitoring window - no error in this case *)
				Done := TRUE;
				iState := STATE_INITIALIZATION;
			END_IF
		END_IF
	ELSE
		(* done after has job false without other monitoring *)
		Done := TRUE;
		iState := STATE_INITIALIZATION;
	END_IF
*)

(* check for timeout *)
ELSIF fbTimeOut.Q THEN
	Error := TRUE;
	ErrorID := MC_ERROR_TARGETPOS_TIMEOUT;
	iState := STATE_INITIALIZATION;
END_IF;
END_ACTION

ACTION ActNcCycleCounter:
(*
	check if cyclic NcToPlc interface changed.
	If not, any Error or CommandAborted condition will be delayed.
	This piece of code prevents from errors if the Plc is called faster than the NC.
	2009-12-08 KSt
*)

fbTimeOutMappingCounter( IN := NcMappingCounter=0, PT:= t#50ms );	(* timout if no nc cyclic feedback for a while *)

NcCycleCounter := DWORD_TO_BYTE(SHR(Axis.NcToPlc.OpModeDWord, 24));
IF NcCycleCounter <> LastNcCycleCounter THEN
	// FAP 04.03.2019 changed from PLC cycles to Nc cycles
	NcMappingCounter := NcMappingCounter + UDINT_TO_BYTE(_F_NcNoOfCycleCounterUpdated(LastNcCycleCounter := LastNcCycleCounter, Axis := Axis)); (* has been reset when the command was initiated *)
//	NcMappingCounter := NcMappingCounter + 1; (* has been reset when the command was initiated *)
	NcCycleCounterAvailable := TRUE; (* marked as available when first time not zero - this flag will never be reset at run-time *)
	NcCycleCounterNotAvailable := FALSE;
ELSIF NOT NcCycleCounterAvailable AND fbTimeOutMappingCounter.Q THEN
	NcCycleCounterNotAvailable := TRUE; (* not available on old target systems *)
END_IF
LastNcCycleCounter:=NcCycleCounter;

// IF NcCycleCounterNotAvailable OR (NcMappingCounter > 1) OR fbTimeOutMappingCounter.Q THEN	// 2017-12-18 KSt
IF NcCycleCounterNotAvailable OR (NcMappingCounter >= 3) OR fbTimeOutMappingCounter.Q THEN		// 2017-12-18 KSt
	(* 	2017-12-18 KSt - wait at least three updates until cyclic data is valid 
	 	two cycles are sufficient on single core systems, three cycles are required on multi core systems
	*)
	(*	NcMappingCounter is set to TRUE after an ADS command has been answered.
		NcCyclicFeedbackExpected is set to TRUE when the NcMappingCounter has been 
		incremented at least twice after an ADS command.
		Also TRUE when cycle counter is not available on old target systems and after a time-out 
	*)
	(* 	If NcCyclicFeedbackExpected is false any wrong condition detected from the
		cyclic NcToPlc interface cannot lead to an Error or CommandAborted result.
	*)
	NcCyclicFeedbackExpected := TRUE;
END_IF
END_ACTION

END_FUNCTION_BLOCK

// POUs/[Internal]/_F_TcMC_IsValidAxisRef
{attribute 'conditionalshow'}
FUNCTION _F_TcMC_IsValidAxisRef : BOOL
VAR_IN_OUT
	Axis : AXIS_REF;
END_VAR
VAR_INPUT
END_VAR
VAR
	TcMemoryArea : E_TcMemoryArea; 
END_VAR

IF __ISVALIDREF(Axis) THEN // AXIS REFERENCE CHECK - 2020-09-17 KSt
	TcMemoryArea := F_CheckMemoryArea(ADR(Axis), SIZEOF(Axis));
	CASE TcMemoryArea OF 
		1 : _F_TcMC_IsValidAxisRef := TRUE;	// static PLC memory
		2 : _F_TcMC_IsValidAxisRef := TRUE;	// dynamic memory
		ELSE
			_F_TcMC_IsValidAxisRef := FALSE;	// invalid
	END_CASE
ELSE
	_F_TcMC_IsValidAxisRef := FALSE;	// invalid
END_IF

END_FUNCTION

// POUs/[Internal]/Axis Status Flag Functions/F_AxisHasExtSetPointGen
{attribute 'conditionalshow'}
FUNCTION F_AxisHasExtSetPointGen : BOOL
(* 	reference: 	NC -> PLC axis interface (128 bytes)
	check if bit 14 of an axis StateDWord is set:
	Axis has an external set point generator (PLC)
	Achse hat einen externen Sollwertgenerator (SPS)
*)
VAR_INPUT
	StateDWord : DWORD;
END_VAR
VAR
END_VAR

F_AxisHasExtSetPointGen := (StateDWord AND 2#0000_0000_0000_0000_0100_0000_0000_0000) <> 0;

END_FUNCTION

// POUs/Motion/Point To Point Motion/MC_Stop
FUNCTION_BLOCK MC_Stop
(*	This FB is primarily intended for emergency stop functionality or exception
	situations.
	This Function Block commands a controlled motion stop and transfers the
	axis to the state 'Stopping'. While the axis is in state Stopping, no other FB 
	can perform any motion on the same axis. After the axis has reached velocity 
	zero, the Done output is set to TRUE immediately. The axis remains in the 
	state 'Stopping' as long as Execute is still TRUE or velocity zero is not yet 
	reached. As soon as 'Done' is set and 'Execute' is FALSE the axis goes to 
	state 'StandStill'.
*)
VAR_IN_OUT
	Axis				:	AXIS_REF; (*Reference to an axis*)
END_VAR
VAR_INPUT
	Execute			:	BOOL;	
	Deceleration		:	LREAL;	
	Jerk				:	LREAL;	
(*	BufferMode		:	MC_BufferMode;*)	 (* 2008-06-27 KSt - deleted after PlcOpen corrigendum V0.4 *)
	Options			: 	ST_MoveOptions; (* optional parameters *)
END_VAR
VAR_OUTPUT
	Done			:	BOOL;	
	Busy			: 	BOOL;	
	Active			: 	BOOL;	
	CommandAborted	:	BOOL;	
	Error			:	BOOL;	
{attribute 'displaymode':='hex'}
	ErrorID			:	UDINT;	
END_VAR
VAR
	LastExecutionResult: 	_ST_FunctionBlockResults;
	ADSbusy		: 	BOOL;
	MoveGeneric		: 	_FB_MoveUniversalGeneric;
	ReleaseLock		: 	ADSWRITE;
	CmdNo			: 	UINT;
	AxisMotionCommandsLocked		: 	BOOL;
	iState			: 	_E_TcMC_STATES := STATE_INITIALIZATION;
	NoJobTimer		: 	TON;
END_VAR
VAR
{attribute 'conditionalshow'}
	fbOnTrigger		: 	R_TRIG;
{attribute 'conditionalshow'}
	CounterMotionCommandsLocked: INT;
END_VAR

fbOnTrigger(CLK:= Execute);

CASE iState OF
STATE_INITIALIZATION:	(* *)
	Busy := FALSE;
	Active := FALSE;
	IF NOT Execute THEN
		Done := FALSE;
		CommandAborted := FALSE;
		Error := FALSE;			(* reset at falling edge of Execute *)
		ErrorID := 0;
	END_IF
    	IF fbOnTrigger.Q THEN
		(* initialize output values *)
		Done := FALSE;
		Busy := TRUE;
		Active := FALSE;
		CommandAborted := FALSE;
		Error := FALSE;
		ErrorID := 0;
		ReleaseLock.WRITE:=FALSE;
		NoJobTimer( IN:=FALSE);	(* 20111209 KSt *)
		iState := STATE_ORDER;
	END_IF

STATE_ORDER :
	(* wait until stop is getting active or axis has stopped for a reason *)
	IF 	MoveGeneric.Active OR
		NOT F_AxisHasJob(Axis.NcToPlc.StateDWord)
		THEN
		Active := TRUE;
		ActStop();
		IF NOT ReleaseLock.BUSY THEN (* may be busy after fast stop retrigger *)
			ReleaseLock.WRITE:=FALSE;
			CounterMotionCommandsLocked := 0;
			iState := STATE_RUNNING;
		END_IF
	ELSIF MoveGeneric.Error OR MoveGeneric.CommandAborted THEN	(* ELSIF added 2009-11-09 KSt *)
		Error := MoveGeneric.Error;
		ErrorID := MoveGeneric.ErrorID;
		CommandAborted := MoveGeneric.CommandAborted; (* KSt 2019-07-01 if an axis is locked by MC_Stop only another MC_Stop can abort this command, therefore no release of is lock shall be done *)
		iState := STATE_INITIALIZATION; (* 2019-12-13 KSt command not accepted or aborted, therefore no unlock of the axis *)

// **** removed 2019-12-13 KSt 	
//		IF F_AxisHasJob(Axis.NcToPlc.StateDWord) AND NOT F_AxisMotionCommandsLocked(Axis.NcToPlc.StateDWord) THEN
//			iState := STATE_INITIALIZATION; (* command not accepted *)
//		ELSIF CommandAborted AND F_AxisMotionCommandsLocked(Axis.NcToPlc.StateDWord) THEN (* KSt 2019-07-01 if an axis is locked by MC_Stop only another MC_Stop can abort this command, therefore no release of is lock shall be done *)
//			iState := STATE_INITIALIZATION; 
//		ELSIF Execute THEN
//			iState := STATE_MOTIONCOMMANDSLOCKED;	(* wait to release after Execute is FALSE *)
//		ELSE
//			ReleaseLock.WRITE := TRUE;	(* release axis if Execute is already FALSE *)
//			iState := STATE_WAITING;
//		END_IF

	END_IF

STATE_RUNNING:  (* wait until axis stands still and Execute is FALSE *)
	(* axis is stopping during this state *)
	IF NOT F_AxisHasJob(Axis.NcToPlc.StateDWord) THEN
		NoJobTimer.IN := TRUE;
	END_IF
//	NoJobTimer( PT:=TcMcGlobal.tStopMonitoringTimeOut + T#50ms );	(* 20111209 KSt - just a safety timer - typically not relevant if MoveGeneric is working correctly *)
  	NoJobTimer( PT:=TcMcGlobal.tStopMonitoringTimeOut + SEL(Options.EnableStopPositionMonitoring AND TcMcGlobal.NcDeviceInfoNcVersion >= 16#03011194 (* NC 4500 *) , T#50MS, TcMcGlobal.tTargetPosTimeOut));	(* 20191016 KSt - just a safety timer - typically not relevant if MoveGeneric is working correctly *)
	IF 	NOT MoveGeneric.Busy OR					(* successfully stopped *)
		(* NOT F_AxisHasJob(Axis.NcToPlc.StateDWord)*) (* or in standstill for any other reason *)	(* 20111209 KSt *)
		NoJobTimer.Q (* or in standstill for any other reason *)	(* 20111209 KSt *)
		THEN
		Error := MoveGeneric.Error;		(* 2008-11-26 KSt *)
		ErrorID := MoveGeneric.ErrorID;	(* 2008-11-26 KSt *)
		CommandAborted := MoveGeneric.CommandAborted;	(* KSt 2009-04-15 *)
		Done := NOT Error AND NOT CommandAborted;		(* KSt 2009-04-15 *)
		(* FAP2019-05-20 if an axis is locked by MC_Stop only another MC_Stop can abort this command, therefore no release of is lock shall be done *)
		IF CommandAborted THEN
			iState := STATE_INITIALIZATION;		
		ELSIF Execute THEN
			iState := STATE_MOTIONCOMMANDSLOCKED;
		ELSE
			ReleaseLock.WRITE := TRUE;	(* release axis if Execute is already FALSE *)
			iState := STATE_WAITING;
		END_IF
	END_IF

STATE_MOTIONCOMMANDSLOCKED : 	(* axis is in standstill and axis is locked against motion commands during this state *)
	IF AxisMotionCommandsLocked AND NOT F_AxisMotionCommandsLocked(Axis.NcToPlc.StateDWord) THEN (* IF block added 2015-03-19 KSt *)
		(* if axis was locked but is not locked anymore it may have been released by a axis reset command *)
		(* IF block added 2015-03-19 KSt *)
		Done := FALSE;
		CommandAborted := NOT Error;
		iState := STATE_INITIALIZATION;
	ELSIF NOT Execute THEN	(* reset outputs if Execute is FALSE *)
		Done := FALSE;
		CommandAborted := FALSE;
		Error := FALSE;
		ErrorID := 0;
		ReleaseLock.WRITE:=TRUE;	(* release axis *)
		CounterMotionCommandsLocked := 0;
		iState := STATE_WAITING;
	END_IF

STATE_WAITING : (* release axis and wait until axis is released *)
	IF NOT Execute THEN	(* reset outputs if Execute is FALSE *)
		Done := FALSE;
		CommandAborted := FALSE;
		Error := FALSE;
		ErrorID := 0;
	END_IF
	ReleaseLock.WRITE:=TRUE;
	ActStop(); (* call here - fast reaction required *)
	IF NOT ReleaseLock.BUSY THEN
		IF ReleaseLock.ERR THEN
			Error := TRUE;
			ErrorID := ReleaseLock.ERRID;
			iState := STATE_INITIALIZATION;
		(* ELSIF NOT F_AxisMotionCommandsLocked(Axis.NcToPlc.StateDWord) THEN *) (* NOT deleted 2009-05-11 KSt *)
		ELSIF F_AxisMotionCommandsLocked(Axis.NcToPlc.StateDWord) THEN
			CounterMotionCommandsLocked := CounterMotionCommandsLocked + 1; (* wait for a certain number of cycles before error - 2009-10-06 KSt *)
			IF CounterMotionCommandsLocked > TcMcGlobal.NCTOPLC_FEEDBACK_MAXWAITCYCLES THEN
				Error := TRUE;
				ErrorID := MC_ERROR_BUFFERED_COMMAND_NO_STATE_FEEDBACK; (* lock bit has not been reset *)
				iState := STATE_INITIALIZATION;
			END_IF
		ELSE (* axis released - no error *)
			iState := STATE_INITIALIZATION;
		END_IF
		ReleaseLock.WRITE:=FALSE;
	END_IF

	IF fbOnTrigger.Q THEN (* KSt 2009-04-15 - Stop retrigger allowed after release even without a "released" feedback*)
		(* initialize output values *)
		Done := FALSE;
		Busy := TRUE;
		Active := FALSE;
		CommandAborted := FALSE;
		Error := FALSE;
		ErrorID := 0;
		ReleaseLock.WRITE:=FALSE;
		iState := STATE_ORDER;	(* retrigger stop command *)
	END_IF

END_CASE

ActStop(); (* call function blocks *)

ADSbusy := MoveGeneric.ADSbusy OR ReleaseLock.BUSY;
IF iState=STATE_INITIALIZATION THEN
	(* reset Busy immediately  when sequence ends *)
	Done:=FALSE;
	Busy := FALSE;
	Active := FALSE;
END_IF

ACTION ActStop:
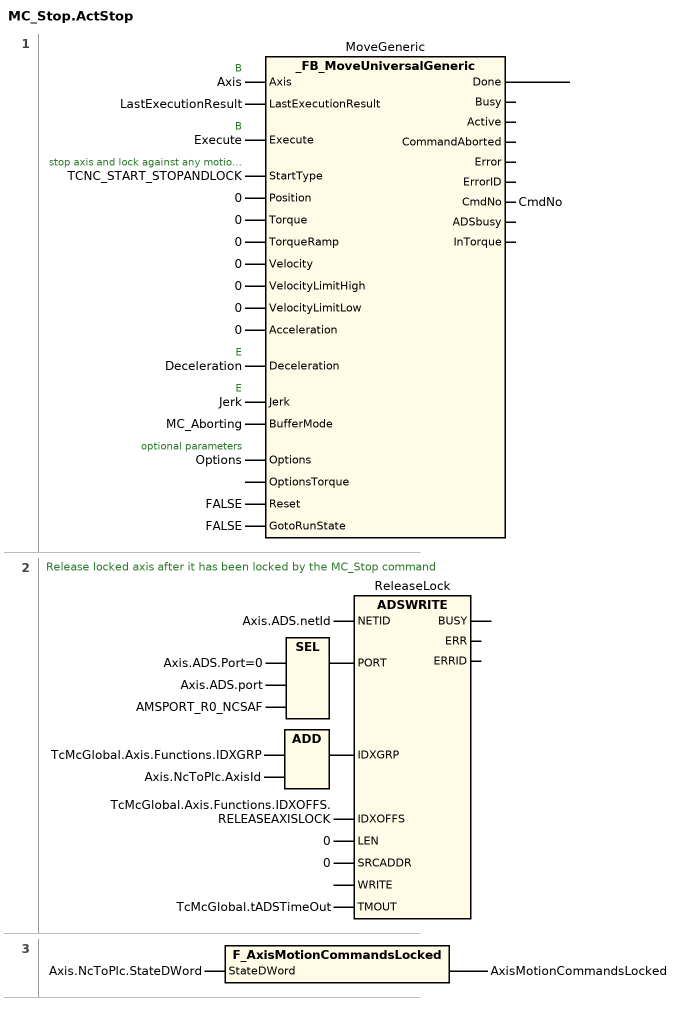
// NETWORK 1
//   Axis: B
//   Execute: B
//   TCNC_START_STOPANDLOCK: stop axis and lock against any motion commands
//   Deceleration: E
//   Jerk: E
//   Options: optional parameters
MoveGeneric(
    Axis := Axis,
    LastExecutionResult := LastExecutionResult,
    Execute := Execute,
    StartType := TCNC_START_STOPANDLOCK,
    Position := 0,
    Torque := 0,
    TorqueRamp := 0,
    Velocity := 0,
    VelocityLimitHigh := 0,
    VelocityLimitLow := 0,
    Acceleration := 0,
    Deceleration := Deceleration,
    Jerk := Jerk,
    BufferMode := MC_Aborting,
    Options := Options,
    Reset := FALSE,
    GotoRunState := FALSE,
    CmdNo => CmdNo); // _FB_MoveUniversalGeneric

// NETWORK 2
// Release locked axis after it has been locked by the MC_Stop command
ReleaseLock(
    NETID := Axis.ADS.netId,
    PORT := SEL(Axis.ADS.Port=0, Axis.ADS.port, AMSPORT_R0_NCSAF),
    IDXGRP := TcMcGlobal.Axis.Functions.IDXGRP + Axis.NcToPlc.AxisId,
    IDXOFFS := TcMcGlobal.Axis.Functions.IDXOFFS.RELEASEAXISLOCK,
    LEN := 0,
    SRCADDR := 0,
    TMOUT := TcMcGlobal.tADSTimeOut); // ADSWRITE

// NETWORK 3
AxisMotionCommandsLocked := F_AxisMotionCommandsLocked(StateDWord := Axis.NcToPlc.StateDWord);
END_ACTION

END_FUNCTION_BLOCK

// POUs/[Internal]/Axis Status Flag Functions/F_AxisMotionCommandsLocked
{attribute 'conditionalshow'}
FUNCTION F_AxisMotionCommandsLocked : BOOL
(* 	reference: 	NC -> PLC axis interface (128 bytes)
	check if bit 29 of an axis StateDWord is set:
	Axis motion commands locked 
	Achse ist gegen Bewegungskommandos gesperrt 
*)
VAR_INPUT
	StateDWord : DWORD;
END_VAR
VAR
END_VAR

F_AxisMotionCommandsLocked := (StateDWord AND 2#0010_0000_0000_0000_0000_0000_0000_0000) <> 0;

END_FUNCTION

// POUs/[Internal]/_F_TcMC_DWORD_TO_HEXSTR
{attribute 'conditionalshow'}
FUNCTION _F_TcMC_DWORD_TO_HEXSTR : STRING(4)
(* convert a decimal number to a hex string *)
VAR_INPUT
	in				: DWORD;
END_VAR
VAR
	str1 : STRING(4);
	pstr: POINTER TO BYTE;
	i: INT;
	digit: BYTE;
END_VAR

str1 := '@@@@';
pstr := ADR(str1) + 4;
FOR i := 1 TO 4 DO
	pstr := pstr - 1;
	digit := DWORD_TO_BYTE(in AND 16#F);
	IF digit < 10 THEN
		digit := digit + 48;
	ELSE
		digit := digit + 65 - 10;
	END_IF
	pstr^ := digit;
	in := in / 16;
END_FOR
_F_TcMC_DWORD_TO_HEXSTR := str1;

END_FUNCTION

// POUs/[Internal]/_F_TcMC_Round
{attribute 'conditionalshow'}
FUNCTION _F_TcMC_Round : LREAL
VAR_INPUT
	value : LREAL;
	digits : BYTE;
END_VAR
VAR
	n: LREAL;
END_VAR

n := EXPT(10, digits);
_F_TcMC_Round := FLOOR(value*n+0.5)/n;

END_FUNCTION

// POUs/Motion/Torque Control/MC_AbortTorqueControl
{attribute 'conditionalshow'}
FUNCTION_BLOCK MC_AbortTorqueControl
VAR_IN_OUT
	Axis						: AXIS_REF;
END_VAR
VAR_INPUT
	Execute						: BOOL;
END_VAR
VAR_OUTPUT
	Done						: BOOL;
	Busy						: BOOL;
	Active						: BOOL;
	CommandAborted				: BOOL;
	Error						: BOOL;
{attribute 'displaymode':='hex'}
	ErrorId						: UDINT;
END_VAR
VAR
	LastExecutionResult: 	_ST_FunctionBlockResults;
	ADSbusy		: 	BOOL;
	MoveGeneric		: 	_FB_MoveUniversalGeneric;
	CmdNo: UINT;
END_VAR

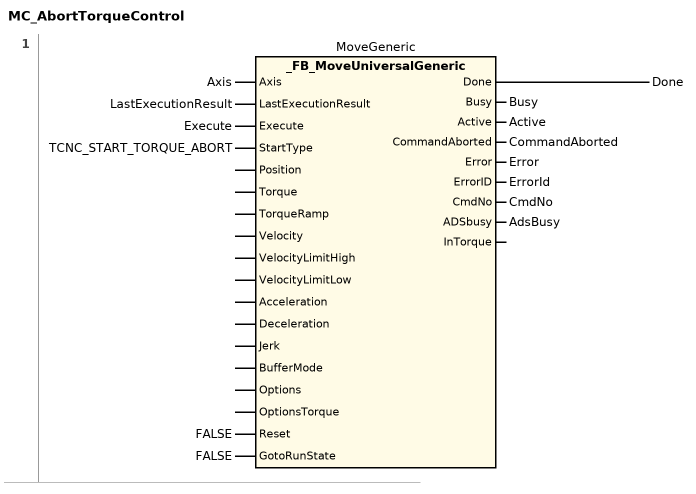
// NETWORK 1
MoveGeneric(
    Axis := Axis,
    LastExecutionResult := LastExecutionResult,
    Execute := Execute,
    StartType := TCNC_START_TORQUE_ABORT,
    Reset := FALSE,
    GotoRunState := FALSE,
    Busy => Busy,
    Active => Active,
    CommandAborted => CommandAborted,
    Error => Error,
    ErrorID => ErrorId,
    CmdNo => CmdNo,
    ADSbusy => AdsBusy); // _FB_MoveUniversalGeneric
Done := MoveGeneric.Done;

END_FUNCTION_BLOCK

// POUs/[Internal]/Axis Status Flag Functions/F_AxisIsMovingEndless
{attribute 'conditionalshow'}
FUNCTION F_AxisIsMovingEndless  : BOOL
(* 	reference: 	NC -> PLC axis interface (128 bytes)
	check if bit 19 of an axis StateDWord is set:
	Axis is moving endless
	Achse in Endlos-Betriebsart
*)
VAR_INPUT
	StateDWord : DWORD;
END_VAR
VAR
END_VAR

F_AxisIsMovingEndless := (StateDWord AND 2#0000_0000_0000_1000_0000_0000_0000_0000) <> 0;

END_FUNCTION

// POUs/[Internal]/Axis Status Flag Functions/F_AxisReachedConstantVelocity
{attribute 'conditionalshow'}
FUNCTION F_AxisReachedConstantVelocity  : BOOL
(* 	reference: 	NC -> PLC axis interface (128 bytes)
	check if bit 12 of an axis StateDWord is set:
	Axis has reached its constant velocity or rotary speed
	Achse hat V-Konst bzw. Drehzahl erreicht
*)
VAR_INPUT
	StateDWord : DWORD;
END_VAR
VAR
END_VAR

F_AxisReachedConstantVelocity := (StateDWord AND 2#0000_0000_0000_0000_0001_0000_0000_0000) <> 0;

END_FUNCTION

// POUs/[Internal]/Axis Status Flag Functions/F_AxisIsCompensating
{attribute 'conditionalshow'}
FUNCTION F_AxisIsCompensating  : BOOL
(* 	reference: 	NC -> PLC axis interface (128 bytes)
	check if bit 13 of an axis StateDWord is set:
 	After a "Distance Compensation" is startet this bit means:
	Axis is in compensation mode
*)
VAR_INPUT
	StateDWord : DWORD;
END_VAR
VAR
END_VAR

F_AxisIsCompensating := (StateDWord AND 2#0000_0000_0000_0000_0010_0000_0000_0000) <> 0;

END_FUNCTION

// POUs/[Internal]/Axis Status Flag Functions/F_AxisDriveLimitActive
{attribute 'conditionalshow'}
FUNCTION F_AxisDriveLimitActive  : BOOL
(* 	reference: 	NC -> PLC axis interface (128 bytes)
	check if bit 15 of an axis StateDWord is set:
	This bit is set while a phasing operation is busy.
	The flag is used at a slave axis of a coupling.
*)
VAR_INPUT
	StateDWord : DWORD;
END_VAR
VAR
END_VAR

F_AxisDriveLimitActive := (StateDWord AND 2#0000_0000_0000_0100_0000_0000_0000_0000) <> 0;

END_FUNCTION

// POUs/Motion/Point To Point Motion/MC_MoveAbsolute
FUNCTION_BLOCK MC_MoveAbsolute
(*	This Function Block commands a controlled motion to a specified absolute position.	*)
VAR_IN_OUT
	Axis				:	AXIS_REF; (*Reference to an axis*)
END_VAR
VAR_INPUT
	Execute			:	BOOL;	(* Start the motion at rising edge *)
(*	ContinuousUpdate :	BOOL; *)		(* not available *)
	Position			:	LREAL;		(* Target position for the motion *)
	Velocity			:	LREAL;		(* Value of the maximum velocity *)
	Acceleration		:	LREAL;		(* Value of the maximum acceleration *)
	Deceleration		:	LREAL;		(* Value of the maximum deceleration *)
	Jerk				:	LREAL;		(* Value of the maximum jerk *)
(*	Direction			:	MC_Direction; *)		(* not available *)
	BufferMode		:	MC_BufferMode;	
	Options			: 	ST_MoveOptions;		(* optional parameters *)
END_VAR
VAR_OUTPUT
	Done			:	BOOL;	
	Busy			: 	BOOL;	
	Active			: 	BOOL;	
	CommandAborted	:	BOOL;	
	Error			:	BOOL;	
{attribute 'displaymode':='hex'}
	ErrorID			:	UDINT;	
END_VAR
VAR
	LastExecutionResult: 	_ST_FunctionBlockResults;
	ADSbusy		: 	BOOL;
	MoveGeneric		: 	_FB_MoveUniversalGeneric;
	CmdNo: UINT;
END_VAR

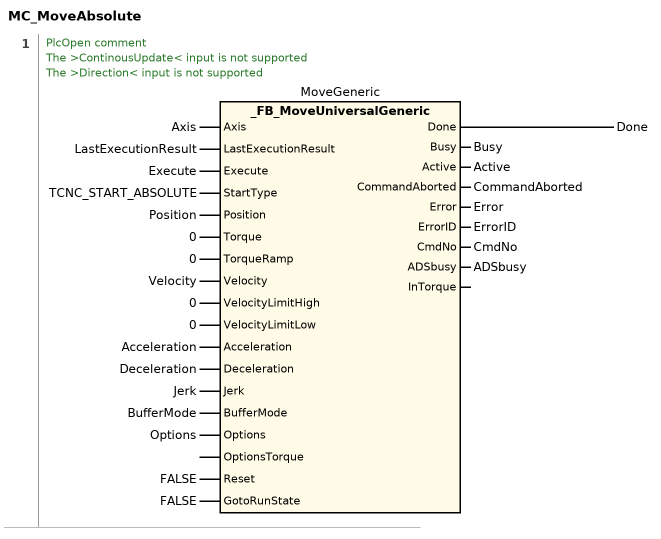
// NETWORK 1
// 					PlcOpen comment
//     The >ContinousUpdate< input is not supported
//     The >Direction< input is not supported
//
//
MoveGeneric(
    Axis := Axis,
    LastExecutionResult := LastExecutionResult,
    Execute := Execute,
    StartType := TCNC_START_ABSOLUTE,
    Position := Position,
    Torque := 0,
    TorqueRamp := 0,
    Velocity := Velocity,
    VelocityLimitHigh := 0,
    VelocityLimitLow := 0,
    Acceleration := Acceleration,
    Deceleration := Deceleration,
    Jerk := Jerk,
    BufferMode := BufferMode,
    Options := Options,
    Reset := FALSE,
    GotoRunState := FALSE,
    Busy => Busy,
    Active => Active,
    CommandAborted => CommandAborted,
    Error => Error,
    ErrorID => ErrorID,
    CmdNo => CmdNo,
    ADSbusy => ADSbusy); // _FB_MoveUniversalGeneric
Done := MoveGeneric.Done;

END_FUNCTION_BLOCK

// POUs/[Internal]/Axis Status Flag Functions/F_AxisIsAtTargetPosition
{attribute 'conditionalshow'}
FUNCTION F_AxisIsAtTargetPosition  : BOOL
(* 	reference: 	NC -> PLC axis interface (128 bytes)
	check if bit 4 of an axis StateDWord is set:
	Axis is at target position (PEH) (physical feedback)
	Achse ist in Zielposition (PEH) (physik. Rückmeldung)
*)
VAR_INPUT
	StateDWord : DWORD;
END_VAR
VAR
END_VAR

F_AxisIsAtTargetPosition := (StateDWord AND 2#0000_0000_0000_0000_0000_0000_0001_0000) <> 0;

END_FUNCTION

// POUs/[Internal]/Axis Status Flag Functions/F_AxisInPositionWindow
{attribute 'conditionalshow'}
FUNCTION F_AxisInPositionWindow : BOOL
(* 	reference: 	NC -> PLC axis interface (128 bytes)
	check if bit 3 of an axis StateDWord is set:
	Axis is in position window (physical feedback)
	Achse ist im Positionsbereichsfenster (physik. Rückmeldung) 
*)
VAR_INPUT
	StateDWord : DWORD;
END_VAR
VAR
END_VAR

F_AxisInPositionWindow := (StateDWord AND 2#0000_0000_0000_0000_0000_0000_0000_1000) <> 0;

END_FUNCTION

// POUs/[Internal]/_F_NcNoOfCycleCounterUpdated
{attribute 'conditionalshow'}
FUNCTION _F_NcNoOfCycleCounterUpdated : UDINT (* returns number of NC cycle counter updates since 4018.15 counter is increased only by one each cycle  *)
VAR_INPUT
	LastNcCycleCounter : UDINT;
END_VAR
VAR_IN_OUT
	Axis : AXIS_REF; (*Reference to an axis*)
END_VAR
VAR
	pData : POINTER TO _InternalAxisRefData;
	NcCycleCounter : UDINT;
END_VAR

(* NC cycle counter will be incremented after NC task updated the NcToPlc data structure *)

NcCycleCounter:= DWORD_TO_UDINT( SHR(Axis.NcToPlc.OpModeDWord, 24) );
IF NcCycleCounter <> LastNcCycleCounter THEN
	IF NOT Axis._internal.NcCycleCounterAvailable THEN
		(* set availability flag when cycle counter changed for the first time *)
		pData := ADR(Axis._internal); (* pointer to internal axis data *)
		pData^.NcCycleCounterAvailable := TRUE;
	END_IF
	IF NcCycleCounter < LastNcCycleCounter THEN
		_F_NcNoOfCycleCounterUpdated := NcCycleCounter + 256 - LastNcCycleCounter;
	ELSIF NcCycleCounter > LastNcCycleCounter THEN
		_F_NcNoOfCycleCounterUpdated := NcCycleCounter - LastNcCycleCounter;
	ELSE
		_F_NcNoOfCycleCounterUpdated := 0;	
	END_IF

ELSIF NOT Axis._internal.NcCycleCounterAvailable AND NcCycleCounter=0 AND LastNcCycleCounter=0 THEN
	(* Nc cycle counter is assumed not to be available if it has never been incremented and is allways zero *)
	(* if axis cycle counter is not available then return TRUE *)
	_F_NcNoOfCycleCounterUpdated := 1;

ELSE
	(* nc cylce counter has not been updated *)
	_F_NcNoOfCycleCounterUpdated := 0;
END_IF

END_FUNCTION

// POUs/[Internal]/Axis Status Flag Functions/F_AxisIsCalibrating
{attribute 'conditionalshow'}
FUNCTION F_AxisIsCalibrating : BOOL
(* 	reference: 	NC -> PLC axis interface (128 bytes)
	check if bit 0 of an axis StateDWord is set:
	Axis is in referencing mode ("Axis being calibrated")
	Achse referenziert ("Achse wird geeicht")
*)
VAR_INPUT
	StateDWord : DWORD;
END_VAR
VAR
END_VAR

F_AxisIsCalibrating := (StateDWord AND 2#0000_0000_0000_0000_0000_1000_0000_0000) <> 0;

END_FUNCTION

// POUs/[Internal]/_F_GetTcAxisObjectId
{attribute 'conditionalshow'}
FUNCTION _F_GetTcAxisObjectId : OTCID
VAR_INPUT
	AxisId			: UDINT;
END_VAR
VAR
END_VAR

IF AxisId <= 0 OR AxisId >= 4096 THEN
	_F_GetTcAxisObjectId := 0;	
ELSE
	_F_GetTcAxisObjectId := 16#05010000 + 16#10 * AxisId;
END_IF

END_FUNCTION

// POUs/[Internal]/ADS/_TcMC_ADSRDWRT
{attribute 'conditionalshow'}
FUNCTION_BLOCK _TcMC_ADSRDWRT (* Extended ADS read/write command *)
(*
 	This function block substitutes the generic ADSRDWRT/EX command.
	This block waits for an update of the cyclic NcToPlc interface after 
	the ADS command has been successfully executed.
*)
VAR_IN_OUT
	Axis 			: 	AXIS_REF; (*Reference to an axis*)
END_VAR
VAR_INPUT
	NETID			:	T_AmsNetId;
	PORT			:	T_AmsPort;
	IDXGRP			:	UDINT;
	IDXOFFS		:	UDINT;
	WRITELEN		:	UDINT;
	READLEN		:	UDINT;
	SRCADDR 		:	PVOID;
	DESTADDR 		:	PVOID;
	WRTRD			:	BOOL;
	TMOUT			:	TIME := DEFAULT_ADS_TIMEOUT;
END_VAR
VAR_OUTPUT
	BUSY			:	BOOL;
	ERR			:	BOOL;
{attribute 'displaymode':='hex'}
	ERRID			:	UDINT;
	COUNT_R		:	UDINT;				(* count of bytes actually read *)
END_VAR
VAR
	fbAdsRdWrt				: 	FW_AdsRdWrt;
	NcCycleCounter			: 	BYTE;
	NcCycleCounterAdsEnd	: 	BYTE;
	UpdateCounter			:	BYTE;
	NoUpdateCounter 		: 	BYTE;	(* used for timeout detection *)
	state: INT;
END_VAR


CASE state OF
 0 :	(* call ADS *)
	fbAdsRdWrt(
		sNetId := NETID,
		nPort := PORT,
		nIdxGrp := IDXGRP,
		nIdxOffs := IDXOFFS,
		cbWriteLen := WRITELEN,
		cbReadLen := READLEN,
		pWriteBuff := SRCADDR,
		pReadBuff := DESTADDR,
		bExecute := WRTRD,
		tTimeout := TMOUT
		);
	IF fbAdsRdWrt.bBusy THEN
		BUSY := TRUE;
		ERR := FALSE;
		ERRID := 0;
		COUNT_R := 0;
		UpdateCounter:=0;
		NoUpdateCounter:=0;
		state := state + 1;
	END_IF

 1 :	(* wait till ADS call is finished *)
	fbAdsRdWrt();
	IF NOT fbAdsRdWrt.bBusy THEN
		IF fbAdsRdWrt.bError THEN
			(* error - feedback without any delay *)
			BUSY := FALSE;
			ERR := fbAdsRdWrt.bError;
			ERRID := fbAdsRdWrt.nErrId;
			COUNT_R := fbAdsRdWrt.cbRead;
			fbAdsRdWrt(bExecute := WRTRD);
			state := 0;
		ELSE
			(* save current NC cycle counter to check for AXIS_REF update in the next state *)
			NcCycleCounter := _F_UpdateNcCycleCounter(Axis);(* store cycle counter at the end of the ADS command sequence *)
			NcCycleCounterAdsEnd := NcCycleCounter;
			state := state + 1;
		END_IF
	END_IF

 2 :	(* wait for AXIS_REF update *)
	IF _F_NcCycleCounterUpdated( LastNcCycleCounter:=NcCycleCounter, Axis:=Axis ) THEN
		UpdateCounter := UpdateCounter + 1;
	ELSE
		NoUpdateCounter:=NoUpdateCounter+1;
		IF NoUpdateCounter>100 THEN
			BUSY := FALSE;
			ERR := TRUE;
			ERRID := MC_ERROR_NCCYCLECOUNTERUPDATE;
			fbAdsRdWrt(bExecute := WRTRD);
			state := 0;
		END_IF
	END_IF
	NcCycleCounter := _F_UpdateNcCycleCounter(Axis);(* store cycle counter when leaving this command *)

	IF UpdateCounter >= 2 THEN	(* at least two updates after response on ADS command *)
		BUSY := FALSE;
		ERR := fbAdsRdWrt.bError;
		ERRID := fbAdsRdWrt.nErrId;
		COUNT_R := fbAdsRdWrt.cbRead;
		fbAdsRdWrt(bExecute := WRTRD);
		state := 0;
	END_IF
END_CASE

END_FUNCTION_BLOCK

// POUs/[Internal]/_F_UpdateNcCycleCounter
{attribute 'conditionalshow'}
FUNCTION _F_UpdateNcCycleCounter : BYTE (* returns NC cycle counter *)
VAR_IN_OUT
	Axis : AXIS_REF; (*Reference to an axis*)
END_VAR

(* NC cycle counter will be incremented after NC task updated the NcToPlc data structure *)

_F_UpdateNcCycleCounter := DWORD_TO_BYTE( SHR(Axis.NcToPlc.OpModeDWord, 24) );

END_FUNCTION

// POUs/[Internal]/_F_NcCycleCounterUpdated
{attribute 'conditionalshow'}
FUNCTION _F_NcCycleCounterUpdated : BOOL (* returns NC cycle counter *)
VAR_INPUT
	LastNcCycleCounter : UDINT;
END_VAR
VAR_IN_OUT
	Axis : AXIS_REF; (*Reference to an axis*)
END_VAR
VAR
	pData : POINTER TO _InternalAxisRefData;
	NcCycleCounter : BYTE;
END_VAR

(* NC cycle counter will be incremented after NC task updated the NcToPlc data structure *)

NcCycleCounter:= DWORD_TO_BYTE( SHR(Axis.NcToPlc.OpModeDWord, 24) );
IF NcCycleCounter <> LastNcCycleCounter THEN
	IF NOT Axis._internal.NcCycleCounterAvailable THEN
		(* set availability flag when cycle counter changed for the first time *)
		pData := ADR(Axis._internal); (* pointer to internal axis data *)
		pData^.NcCycleCounterAvailable := TRUE;
	END_IF
	_F_NcCycleCounterUpdated := TRUE;

ELSIF NOT Axis._internal.NcCycleCounterAvailable AND NcCycleCounter=0 AND LastNcCycleCounter=0 THEN
	(* Nc cycle counter is assumed not to be available if it has never been incremented and is allways zero *)
	(* if axis cycle counter is not available then return TRUE *)
	_F_NcCycleCounterUpdated := TRUE;

ELSE
	(* nc cylce counter has not been updated *)
	_F_NcCycleCounterUpdated := FALSE;
END_IF

END_FUNCTION

// POUs/[Internal]/ADS/_TcMC_ADSREAD
{attribute 'conditionalshow'}
FUNCTION_BLOCK _TcMC_ADSREAD (* Extended ADS read command *)
(*
 	This function block substitutes the generic ADSREAD/EX command.
	This block waits for an update of the cyclic NcToPlc interface after 
	the ADS command has been successfully executed.
*)
VAR_IN_OUT
	Axis 			: 	AXIS_REF; (*Reference to an axis*)
END_VAR
VAR_INPUT
	NETID			:	T_AmsNetId;
	PORT			:	T_AmsPort;
	IDXGRP			:	UDINT;
	IDXOFFS		:	UDINT;
	LEN				:	UDINT;
	DESTADDR 		:	PVOID;
	READ			:	BOOL;
	TMOUT			:	TIME := DEFAULT_ADS_TIMEOUT;
END_VAR
VAR_OUTPUT
	BUSY			:	BOOL;
	ERR			:	BOOL;
{attribute 'displaymode':='hex'}
	ERRID			:	UDINT;
	COUNT_R		:	UDINT;	(* count of bytes actually read *)
END_VAR
VAR
	fbAdsRead				: 	FW_AdsRead;
	NcCycleCounter			: 	BYTE;
	NcCycleCounterAdsEnd	: 	BYTE;
	UpdateCounter			:	BYTE;
	NoUpdateCounter 		: 	BYTE;	(* used for timeout detection *)
	state: INT;
END_VAR


CASE state OF
 0 :	(* call ADS *)
	fbAdsRead(
		sNetId := NETID,
		nPort := PORT,
		nIdxGrp := IDXGRP,
		nIdxOffs := IDXOFFS,
		cbReadLen := LEN,
		pReadBuff := DESTADDR,
		bExecute := READ,
		tTimeout := TMOUT
		);
	IF fbAdsRead.bBusy THEN
		BUSY := TRUE;
		ERR := FALSE;
		ERRID := 0;
		COUNT_R := 0;
		UpdateCounter:=0;
		NoUpdateCounter:=0;
		state := state + 1;
	END_IF

 1 :	(* wait till ADS call is finished *)
	fbAdsRead();
	IF NOT fbAdsRead.bBusy THEN
		IF fbAdsRead.bError THEN
			(* error - feedback without any delay *)
			BUSY := FALSE;
			ERR := fbAdsRead.bError;
			ERRID := fbAdsRead.nErrId;
			COUNT_R := fbAdsRead.cbRead;
			fbAdsRead(bExecute := READ);
			state := 0;
		ELSE
			(* save current NC cycle counter to check for AXIS_REF update in the next state *)
			NcCycleCounter := _F_UpdateNcCycleCounter(Axis);(* store cycle counter at the end of the ADS command sequence *)
			NcCycleCounterAdsEnd := NcCycleCounter;
			state := state + 1;
		END_IF
	END_IF

 2 :	(* wait for AXIS_REF update *)
	IF _F_NcCycleCounterUpdated( LastNcCycleCounter:=NcCycleCounter, Axis:=Axis ) THEN
		UpdateCounter := UpdateCounter + 1;
	ELSE
		NoUpdateCounter:=NoUpdateCounter+1;
		IF NoUpdateCounter>100 THEN
			BUSY := FALSE;
			ERR := TRUE;
			ERRID := MC_ERROR_NCCYCLECOUNTERUPDATE;
			fbAdsRead(bExecute := READ);
			state := 0;
		END_IF
	END_IF
	NcCycleCounter := _F_UpdateNcCycleCounter(Axis);(* store cycle counter when leaving this command *)

	IF UpdateCounter >= 2 THEN	(* at least two updates after response on ADS command *)
		BUSY := FALSE;
		ERR := fbAdsRead.bError;
		ERRID := fbAdsRead.nErrId;
		COUNT_R := fbAdsRead.cbRead;
		fbAdsRead(bExecute := READ);
		state := 0;
	END_IF
END_CASE

END_FUNCTION_BLOCK

// POUs/[Internal]/ADS/_TcMC_ADSWRITE
{attribute 'conditionalshow'}
FUNCTION_BLOCK _TcMC_ADSWRITE (* ADS write command *)
(*
 	This function block substitutes the generic ADSWRITE command.
	This block waits for an update of the cyclic NcToPlc interface after 
	the ADS command has been successfully executed.
*)
VAR_IN_OUT
	Axis 			: 	AXIS_REF; (*Reference to an axis*)
END_VAR
VAR_INPUT
	NETID			:	T_AmsNetId;
	PORT			:	T_AmsPort;
	IDXGRP			:	UDINT;
	IDXOFFS		:	UDINT;
	LEN				:	UDINT;
	SRCADDR 		:	PVOID;
	WRITE			:	BOOL;
	TMOUT			:	TIME := DEFAULT_ADS_TIMEOUT;
END_VAR
VAR_OUTPUT
	BUSY			:	BOOL;
	ERR			:	BOOL;
{attribute 'displaymode':='hex'}
	ERRID			:	UDINT;
END_VAR
VAR
	fbAdsWrite				: 	FW_AdsWrite;
	NcCycleCounter			: 	BYTE;
	NcCycleCounterAdsEnd	: 	BYTE;
	UpdateCounter			:	BYTE;
	NoUpdateCounter 		: 	BYTE;	(* used for timeout detection *)
	state: INT;
END_VAR


CASE state OF
 0 :	(* call ADS *)
	fbAdsWrite(
		sNetId := NETID,
		nPort := PORT,
		nIdxGrp := IDXGRP,
		nIdxOffs := IDXOFFS,
		cbWriteLen := LEN,
		pWriteBuff := SRCADDR,
		bExecute := WRITE,
		tTimeout := TMOUT
		);
	IF fbAdsWrite.bBusy THEN
		BUSY := TRUE;
		ERR := FALSE;
		ERRID := 0;
		UpdateCounter:=0;
		NoUpdateCounter:=0;
		state := state + 1;
	END_IF

 1 :	(* wait till ADS call is finished *)
	fbAdsWrite();
	IF NOT fbAdsWrite.bBusy THEN
		IF fbAdsWrite.bError THEN
			(* error - feedback without any delay *)
			BUSY := FALSE;
			ERR := fbAdsWrite.bError;
			ERRID := fbAdsWrite.nErrId;
			fbAdsWrite(bExecute := WRITE);
			state := 0;
		ELSE
			(* save current NC cycle counter to check for AXIS_REF update in the next state *)
			NcCycleCounter := _F_UpdateNcCycleCounter(Axis);(* store cycle counter at the end of the ADS command sequence *)
			NcCycleCounterAdsEnd := NcCycleCounter;
			state := state + 1;
		END_IF
	END_IF

 2 :	(* wait for AXIS_REF update *)
	IF _F_NcCycleCounterUpdated( LastNcCycleCounter:=NcCycleCounter, Axis:=Axis ) THEN
		UpdateCounter := UpdateCounter + 1;
	ELSE
		NoUpdateCounter:=NoUpdateCounter+1;
		IF NoUpdateCounter>100 THEN
			BUSY := FALSE;
			ERR := TRUE;
			ERRID := MC_ERROR_NCCYCLECOUNTERUPDATE;
			fbAdsWrite(bExecute := WRITE);
			state := 0;
		END_IF
	END_IF
	NcCycleCounter := _F_UpdateNcCycleCounter(Axis);(* store cycle counter when leaving this command *)

	IF UpdateCounter >= 2 THEN	(* at least two updates after response on ADS command *)
		BUSY := FALSE;
		ERR := fbAdsWrite.bError;
		ERRID := fbAdsWrite.nErrId;
		fbAdsWrite(bExecute := WRITE);
		state := 0;
	END_IF
END_CASE

END_FUNCTION_BLOCK

// POUs/[Internal]/Axis Status Flag Functions/F_AxisCamDataQueued
{attribute 'conditionalshow'}
FUNCTION F_AxisCamDataQueued : BOOL
(* 	reference: 	NC -> PLC axis interface (128 bytes)
	check if bit 22 of an axis StateDWord is set:
	New cam data has been queued to a slave axis which is coupled to master via a cam table. 
	The flag comes up when the PLC modifies the camming data.
	Das Flag wird TRUE, wenn neue bzw. veränderte Kurvenscheibendaten von der SPS an 
	eine Slave-Achse gesendet werden.
*)
VAR_INPUT
	StateDWord : DWORD;
END_VAR
VAR
END_VAR

F_AxisCamDataQueued := (StateDWord AND 2#0000_0000_0100_0000_0000_0000_0000_0000) <> 0;

END_FUNCTION

// POUs/[Internal]/Axis Status Flag Functions/F_AxisCamScalingPending
{attribute 'conditionalshow'}
FUNCTION F_AxisCamScalingPending : BOOL
(* 	reference: 	NC -> PLC axis interface (128 bytes)
	check if bit 23 of an axis StateDWord is set:
	- The flag signals that the scaling and/or offset setting of a cam table has been requested 
	to be performed 	at a certain master position. This request is pending while the function 
	result is TRUE and has been executed after a falling edge of this signal.
	- Das Flag zeigt an das die Skalierung und/oder das Setzen der Offsets einer Kurvenscheibe
	beauftrag wurde aber erst später (ab einer bestimmten Master-Position) durchgeführt wird.
	Mit fallender Flanke des Signals wurde der Auftrag ausgeführt.
*)
VAR_INPUT
	StateDWord : DWORD;
END_VAR
VAR
END_VAR

F_AxisCamScalingPending := (StateDWord AND 2#0000_0000_1000_0000_0000_0000_0000_0000) <> 0;

END_FUNCTION

// POUs/[Internal]/Axis Status Flag Functions/F_AxisCamTableQueued
{attribute 'conditionalshow'}
FUNCTION F_AxisCamTableQueued : BOOL
(* 	reference: 	NC -> PLC axis interface (128 bytes)
	check if bit 21 of an axis StateDWord is set:
	New cam data has been queued to a slave axis which is coupled to master via a cam table. 
	The flag comes up when the PLC modifies the camming data.
	Das Flag wird TRUE, wenn neue bzw. veränderte Kurvenscheibendaten von der SPS an 
	eine Slave-Achse gesendet werden.
*)
VAR_INPUT
	StateDWord : DWORD;
END_VAR
VAR
END_VAR

F_AxisCamTableQueued := (StateDWord AND 2#0000_0000_0010_0000_0000_0000_0000_0000) <> 0;

END_FUNCTION

// POUs/[Internal]/Axis Status Flag Functions/F_AxisExternalLatchValid
{attribute 'conditionalshow'}
FUNCTION F_AxisExternalLatchValid : BOOL
(* 	reference: 	NC -> PLC axis interface (128 bytes)
	check if bit 16 of an axis StateDWord is set:
	External latch value or sensing switch has become valid
	Externer Latchwert bzw. Messtaster gültig geworden
*)
VAR_INPUT
	StateDWord : DWORD;
END_VAR
VAR
END_VAR

F_AxisExternalLatchValid := (StateDWord AND 2#0000_0000_0000_0001_0000_0000_0000_0000) <> 0;

END_FUNCTION

// POUs/[Internal]/Axis Status Flag Functions/F_AxisGotNewTargetPosition
{attribute 'conditionalshow'}
FUNCTION F_AxisGotNewTargetPosition  : BOOL
(* 	reference: 	NC -> PLC axis interface (128 bytes)
	check if bit 17 of an axis StateDWord is set:
	Axis got a new target position or a new velocity
	while the current move command is in execution.
	Die Zielposition oder die Geschwindigkeit der Achse
	wurde geändert, während die Achse eine Bewegung ausführt
*)
VAR_INPUT
	StateDWord : DWORD;
END_VAR
VAR
END_VAR

F_AxisGotNewTargetPosition := (StateDWord AND 2#0000_0000_0000_0010_0000_0000_0000_0000) <> 0;

END_FUNCTION

// POUs/[Internal]/Axis Status Flag Functions/F_AxisIoDataIsInvalid
{attribute 'conditionalshow'}
FUNCTION F_AxisIoDataIsInvalid : BOOL
(* 	reference: 	NC -> PLC axis interface (128 bytes)
	check if bit 30 of an axis StateDWord is set:
	Axis I/O data is invalid  (e.g. invalid 'WcState' or 'CdlState' )
	Achse hat keine gültigen I/O-Daten  (e.g. invalid 'WcState' or 'CdlState' )
*)
VAR_INPUT
	StateDWord : DWORD;
END_VAR
VAR
END_VAR

F_AxisIoDataIsInvalid := (StateDWord AND 2#0100_0000_0000_0000_0000_0000_0000_0000) <> 0;

END_FUNCTION

// POUs/[Internal]/Axis Status Flag Functions/F_AxisIsCalibrated
{attribute 'conditionalshow'}
FUNCTION F_AxisIsCalibrated : BOOL
(* 	reference: 	NC -> PLC axis interface (128 bytes)
	check if bit 1 of an axis StateDWord is set:
	Axis has been referenced ("Axis calibrated")
	Achse ist referenziert ("Achse geeicht")
*)
VAR_INPUT
	StateDWord : DWORD;
END_VAR
VAR
END_VAR

F_AxisIsCalibrated := (StateDWord AND 2#0000_0000_0000_0000_0000_0000_0000_0010) <> 0;

END_FUNCTION

// POUs/[Internal]/Axis Status Flag Functions/F_AxisIsMoving
{attribute 'conditionalshow'}
FUNCTION F_AxisIsMoving : BOOL
(* 	reference: 	NC -> PLC axis interface (128 bytes)
	check if bit 9 OR 10 of an axis StateDWord is set:
	Axis moving (forward or backwards)
	Achse fährt (vorwärts oder rückwärts)
*)
VAR_INPUT
	StateDWord : DWORD;
END_VAR
VAR
END_VAR

F_AxisIsMoving := (StateDWord AND 2#0000_0000_0000_0000_0000_0110_0000_0000) <> 0;

END_FUNCTION

// POUs/[Internal]/Axis Status Flag Functions/F_AxisIsMovingBackwards
{attribute 'conditionalshow'}
FUNCTION F_AxisIsMovingBackwards : BOOL
(* 	reference: 	NC -> PLC axis interface (128 bytes)
	check if bit 10 of an axis StateDWord is set:
	Axis moving to logically smaller values
	Achse fährt logisch kleiner
*)
VAR_INPUT
	StateDWord : DWORD;
END_VAR
VAR
END_VAR

F_AxisIsMovingBackwards := (StateDWord AND 2#0000_0000_0000_0000_0000_0100_0000_0000) <> 0;

END_FUNCTION

// POUs/[Internal]/Axis Status Flag Functions/F_AxisIsMovingForward
{attribute 'conditionalshow'}
FUNCTION F_AxisIsMovingForward : BOOL
(* 	reference: 	NC -> PLC axis interface (128 bytes)
	check if bit 9 of an axis StateDWord is set:
	Axis moving to logically larger values
	Achse fährt logisch größer
*)
VAR_INPUT
	StateDWord : DWORD;
END_VAR
VAR
END_VAR

F_AxisIsMovingForward := (StateDWord AND 2#0000_0000_0000_0000_0000_0010_0000_0000) <> 0;

END_FUNCTION

// POUs/[Internal]/Axis Status Flag Functions/F_AxisIsNotMoving
{attribute 'conditionalshow'}
FUNCTION F_AxisIsNotMoving : BOOL
(* 	reference: 	NC -> PLC axis interface (128 bytes)
	check if bit 2 of an axis StateDWord is set:
	Axis is logically stationary ("Axis not moving")
	Achse ist im logischen Stillstand ("Achse fährt nicht")
*)
VAR_INPUT
	StateDWord : DWORD;
END_VAR
VAR
END_VAR

F_AxisIsNotMoving := (StateDWord AND 2#0000_0000_0000_0000_0000_0000_0000_0100) <> 0;

END_FUNCTION

// POUs/[Internal]/Axis Status Flag Functions/F_AxisJobPending
{attribute 'conditionalshow'}
FUNCTION F_AxisJobPending : BOOL
(* 	reference: 	NC -> PLC axis interface (128 bytes)
	check if bit 24 of an axis StateDWord is set:
	- The flag signals that the a new motion job ist pending and will be 
	   executed after the active job is finished (buffer mode)
	- Das Flag zeigt an das die ein neuer Fahrauftrag gepuffert ist,
	   um nach dem aktuellen Auftrag ausgeführt zu werden (buffer mode)
*)
VAR_INPUT
	StateDWord : DWORD;
END_VAR
VAR
END_VAR

F_AxisJobPending := (StateDWord AND 2#0000_0001_0000_0000_0000_0000_0000_0000) <> 0;

END_FUNCTION

// POUs/[Internal]/Axis Status Flag Functions/F_AxisPhasingActive
{attribute 'conditionalshow'}
FUNCTION F_AxisPhasingActive  : BOOL
(* 	reference: 	NC -> PLC axis interface (128 bytes)
	check if bit 15 of an axis StateDWord is set:
	This bit is set while a phasing operation is busy.
	The flag is used at a slave axis of a coupling.
*)
VAR_INPUT
	StateDWord : DWORD;
END_VAR
VAR
END_VAR

F_AxisPhasingActive := (StateDWord AND 2#0000_0000_0000_0000_1000_0000_0000_0000) <> 0;

END_FUNCTION

